// NETWORK 2
fbCase_DuplicateUpdateToDB(
    bExecute := bExecute,
    bUseInterimCodeForValidation := bUseInterimCodeForValidation,
    aOCVPackStatus := aOCVPackStatus,
    aOuterStatus := aOuterStatus,
    stOCVDataDB := stOCVDataDB,
    stOACDataDB := stOACDataDB,
    stOuterBarcodeDuplicate := stOuterBarcodeDuplicate,
    stOuterDuplicatedPackCodesFound := stOuterDuplicatedPackCodesFound,
    stCodeInfo_Pack := stCodeInfo_Pack,
    stCodeInfo_Intermediate := stCodeInfo_Intermediate,
    stCodeInfo_Outer := stCodeInfo_Outer,
    stCACData := stCACData,
    bBusy => bBusy,
    bError => bError,
    nErrorID => nErrorID,
    nOACFilesBlocked => nOACFilesBlocked,
    nOCVFilesBlocked => nOCVFilesBlocked,
    stDaigOACDataDB => stDaigOACDataDB,
    stDiagOCVDataDB => stDiagOCVDataDB); // FB_CASE_DuplicateUpdateToDB
bDone := fbCase_DuplicateUpdateToDB.bDone;

ACTION Init:

rTrigDataInit(CLK := bDataInit);

IF rTrigDataInit.Q THEN
	
	stProductInstruction.nOutersPerCase		:= 50;
	stProductInstruction.nPacksPerOuter 	:= 10;
	
	stCACData.NumberOfOuters	:= 50;
	

	FOR iOuter := 1 TO stProductInstruction.nOutersPerCase DO
		(* Ustaw outer *)
		stCACData.Outer[iOuter].Barcode    := CONCAT('OUTER', INT_TO_STRING(iOuter));
		stCACData.Outer[iOuter].OuterCodeStatus := 5;
		
		stCACData.Outer[iOuter].OuterRejectID	:= 0;
		
		
		FOR iPack := 1 TO stProductInstruction.nPacksPerOuter DO
			(* Pack number z zerami *)
			sPackNum := CONCAT('0', INT_TO_STRING(iPack));  (* dla 1-9: '01'-'09' *)
			IF iPack = 10 THEN
				sPackNum := '10';
			END_IF;
			
			(* Outer number z zerami dla 1-9 *)
			sOuterNum := CONCAT('0', INT_TO_STRING(iOuter));
			IF iOuter >= 10 THEN
				sOuterNum := INT_TO_STRING(iOuter);
			END_IF;
			
			(* Sklej pack code *)
			sPackCode := CONCAT(CONCAT('PACK', sPackNum), CONCAT('OUTER', sOuterNum));
			
			(* Przypisz *)
			stCACData.Outer[iOuter].PackCode[iPack]			:= sPackCode;
			stCACData.Outer[iOuter].PackCodeStatus[iPack]	:= 5;
			stCACData.Outer[iOuter].PackRejectID[iPack]		:= 0;
			
		END_FOR;
	END_FOR;	
	
END_IF
END_ACTION

END_PROGRAM

// ---- POUs/FinaliseCaseData/FB_CASE_DuplicateUpdateToDB.TcPOU
(* reads CAC files from CAC folder, deletes OAC file and copies CAC file into Archive *)
FUNCTION_BLOCK FB_CASE_DuplicateUpdateToDB
VAR_INPUT
	bExecute				: BOOL;		(* set TRUE to archive OAC files *)
	bUseInterimCodeForValidation	: BOOL;
END_VAR
VAR_IN_OUT
	
	aOCVPackStatus			: ARRAY[1..cMAX_OUTER_STATUS_QUEUE] OF ST_OUTER_Status;	(* Outer status array *)
	aOuterStatus				: ARRAY[1..cMAX_OUTER_STATUS_QUEUE] OF ST_OUTER_Status;	(* Outer status array *)
	
	//stProductInstruction		: ST_PCM_Status;
	stOCVDataDB				: ST_DB_OCVDataCtrl;
	stOACDataDB				: ST_DB_OACDataCtrl;
	
	stOuterBarcodeDuplicate			: ST_RejectItems;
	stOuterDuplicatedPackCodesFound	: ST_RejectItems;
	
	stCodeInfo_Pack			: ST_CodeInfo;
	stCodeInfo_Intermediate	: ST_CodeInfo;
	stCodeInfo_Outer		: ST_CodeInfo;
	
	stCACData			: ST_CAC_Data;
END_VAR
VAR_OUTPUT
	bDone 					: BOOL;		(* TRUE = OAC archive complete *)
	bBusy 					: BOOL;		(* TRUE = OAC archive active *)
	bError 					: BOOL;		(* TRUE = OAC archive error *)
	nErrorID				: UDINT;	(* error code *)

	nOACFilesBlocked		: UINT;
	nOCVFilesBlocked		: UINT;
	stDaigOACDataDB				: ST_DB_OACDataCtrl;
	stDiagOCVDataDB				: ST_DB_OCVDataCtrl;
	

END_VAR
VAR
	fbExecute				: R_TRIG;
	eState					: E_CAC_State;
	eErrorState				: E_CAC_State;

	tonTimeOut				: TON;
	rtTimeOutExec			: R_TRIG;
	
	stOCVStatus				: ST_OUTER_Status;
	stOACStatus				: ST_OUTER_Status;
	
	nOuterIndex				: INT;
	nOACIndex				: INT;
	nOCVIndex				: INT;
END_VAR

(***************************************TimeOut *******************************************)
(* monitor Busy timeout *)
tonTimeOut( IN:=bBusy, PT:=cTEN_SECONDS, Q=>);
(*	cTHREE_SECONDS						: TIME := T#3s;
	cFIVE_SECONDS						: TIME := t#5s;
	cTEN_SECONDS						: TIME := t#10s;*)

rtTimeOutExec(CLK:= tonTimeOut.Q);

IF rtTimeOutExec.Q THEN

	bError := TRUE;
	nErrorID := 100;
	eErrorState := eState;

	MEMSET(ADR(stOCVDataDB), 16#00, SIZEOF(stOCVDataDB));
	MEMSET(ADR(stOACDataDB), 16#00, SIZEOF(stOACDataDB));

	eState := E_CAC_DONE;
END_IF

(***************************************Execution*******************************************)

(* monitor bExecute for rising edge *)
fbExecute(CLK := bExecute);

CASE eState OF

	(* idle *)
	E_CAC_IDLE:

		(* rising edge of bExecute *)
		IF fbExecute.Q = TRUE THEN

			(* update outputs *)
			bDone := FALSE;
			bBusy := TRUE;
			bError := FALSE;
			nErrorID := 0;

			
			MEMSET(ADR(stOCVDataDB), 16#00, SIZEOF(stOCVDataDB));
			MEMSET(ADR(stOACDataDB), 16#00, SIZEOF(stOACDataDB));

			nOACFilesBlocked 	:= 0;
			nOCVFilesBlocked 	:= 0;

			nOuterIndex			:= 1;
			
			eState := E_CAC_DUPLICATEOUTERCHECK;

		(* bExecute has been reset *)
		ELSIF bExecute = FALSE THEN

			(* clear outputs *)
			bDone := FALSE;
			bBusy := FALSE;
			bError := FALSE;
			(*nErrorID := 0;*)
		END_IF

(*****************************************************************************************)

	(* check outer reject code for dupicate found*)
	E_CAC_DUPLICATEOUTERCHECK:

		IF stCACData.Outer[nOuterIndex].OuterRejectID = stOuterDuplicatedPackCodesFound.nRejectID OR 
			stCACData.Outer[nOuterIndex].OuterRejectID = stOuterBarcodeDuplicate.nRejectID THEN
		
			FillInDBData();
	
			stOACDataDB.bBlockRecord			:= TRUE;
			stOCVDataDB.bBlockRecord			:= TRUE;
			
			stOACDataDB.bUpdateDataReq			:= TRUE;
			stOCVDataDB.bUpdateDataReq			:= TRUE;
			
			eState := E_CAC_DELETEOAC;
		ELSE
			IF nOuterIndex = stCACData.NumberOfOuters THEN

				eState := E_CAC_DONE;
			ELSE
				nOuterIndex := LIMIT(1, nOuterIndex + 1, stCACData.NumberOfOuters);
			END_IF
		END_IF

	(* delete OAC files *)
	E_CAC_DELETEOAC:

		FOR nOACIndex := 1 TO cMAX_OUTER_STATUS_QUEUE DO
			IF aOuterStatus[nOACIndex].stOACData.Barcode =  stOACDataDB.stOACStatusDB.stOACData.Barcode AND 
				aOuterStatus[nOACIndex].stOACData.Barcode <> '' THEN

				//MEMSET(ADR(aOuterStatus[nOACIndex].stOACData), 16#00, SIZEOF(aOuterStatus[nOACIndex].stOACData));
				aOuterStatus[nOACIndex].nStatus.22 := TRUE;
				aOuterStatus[nOACIndex].stOACData.DataSource := 'REM';
			END_IF
		END_FOR

		IF	stOACDataDB.bDone	THEN

			IF NOT  stOACDataDB.bError THEN

				nOACFilesBlocked := nOACFilesBlocked + 1;
			ELSE
				bError := TRUE;
				nErrorID := stOACDataDB.nErrorID;
				eErrorState := eState;
			END_IF
			stDaigOACDataDB := stOACDataDB;
			MEMSET(ADR(stOACDataDB), 16#00, SIZEOF(stOACDataDB));

			eState := E_CAC_DELETEOCV1;
		END_IF

	E_CAC_DELETEOCV1:

		IF stOCVDataDB.stOCVStatusDB.stOACData.AggregationCodes[1] <> '' 	OR 
			stOCVDataDB.stOCVStatusDB.stOACData.AggregationCodes[2] <> '' 	THEN

			FOR nOCVIndex := 1 TO cMAX_OUTER_STATUS_QUEUE DO
				IF aOCVPackStatus[nOCVIndex].stOACData.AggregationCodes[1] =  stOCVDataDB.stOCVStatusDB.stOACData.AggregationCodes[1] 	AND
					aOCVPackStatus[nOCVIndex].stOACData.AggregationCodes[2] =  stOCVDataDB.stOCVStatusDB.stOACData.AggregationCodes[2]	THEN
					
					//MEMSET(ADR(aOCVPackStatus[nOCVIndex].stOACData), 16#00, SIZEOF(aOCVPackStatus[nOCVIndex].stOACData));
					aOCVPackStatus[nOCVIndex].nStatus.22 := TRUE;
					aOCVPackStatus[nOCVIndex].stOACData.DataSource := 'REM';
				END_IF
			END_FOR
		END_IF
		
		IF	stOCVDataDB.bDone	THEN

			IF NOT  stOCVDataDB.bError THEN

				nOCVFilesBlocked := nOCVFilesBlocked + 1;
			ELSE
				bError := TRUE;
				nErrorID := stOCVDataDB.nErrorID;
				eErrorState := eState;
			END_IF

			stDiagOCVDataDB := stOCVDataDB;
			MEMSET(ADR(stOCVDataDB), 16#00, SIZEOF(stOCVDataDB));
			
			IF nOuterIndex = stCACData.NumberOfOuters THEN

				eState := E_CAC_DONE;
			ELSE
				nOuterIndex := LIMIT(1, nOuterIndex + 1, stCACData.NumberOfOuters);
				
				eState := E_CAC_DUPLICATEOUTERCHECK;
			END_IF
		END_IF

	(* complete *)
	E_CAC_DONE:

		(* update outputs *)
		bBusy := FALSE;
		bDone := TRUE;

		eState := E_CAC_IDLE;

(* unknown state *)
ELSE

	eState := E_CAC_IDLE;
END_CASE

ACTION FillInDBData:
(************************************************************Fill In OAC Data****************************************************************************)

IF F_InvalidateASCIIChar(F_CODE_GetItem(stCACData.Outer[nOuterIndex].Barcode, eCodeAIType.SerialCode, stCodeInfo_Outer)) >	0 	THEN

	stOACDataDB.sFileCodeName	:='';
ELSE
	stOACDataDB.sFileCodeName	:= F_CodeToHex(F_CODE_GetItem(stCACData.Outer[nOuterIndex].Barcode , eCodeAIType.SerialCode, stCodeInfo_Outer));
END_IF

stOACDataDB.stOACStatusDB.stOACData	:= stCACData.Outer[nOuterIndex];
stOACDataDB.stOACStatusDB.stOACData.DataSource := 'REM';
stOACDataDB.stOACStatusDB.nTriggerID :=9999;
stOACDataDB.stOACStatusDB.nStatus.22 := TRUE;
stOACDataDB.stOACStatusDB.sDataSourceTracker := 'Dup Update';

FOR nOCVindex :=1 TO stOACDataDB.stOACStatusDB.stOACData.NumberOfPacks DO

	IF	stOACDataDB.stOACStatusDB.stOACData.PackCodeStatus[nOCVindex].5  THEN
		stOACDataDB.stOACStatusDB.aOACPackStatus[nOCVindex] :=5;
	ELSIF stOACDataDB.stOACStatusDB.stOACData.PackCodeStatus[nOCVindex].3  THEN
		stOACDataDB.stOACStatusDB.aOACPackStatus[nOCVindex] :=3;
	ELSE
		stOACDataDB.stOACStatusDB.aOACPackStatus[nOCVindex] :=0;
	END_IF
END_FOR

(************************************************************Fill In OCV Data****************************************************************************)


IF F_InvalidateASCIIChar(F_CODE_GetItem(stCACData.Outer[nOuterIndex].AggregationCodes[1] , eCodeAIType.SerialCode,
										SEL(bUseInterimCodeForValidation, stCodeInfo_Pack, stCodeInfo_Intermediate))) >	0 	THEN

	stOCVDataDB.sFileCodeName1	:= '';
ELSE
	stOCVDataDB.sFileCodeName1	:= F_CodeToHex(F_CODE_GetItem(stCACData.Outer[nOuterIndex].AggregationCodes[1] , eCodeAIType.SerialCode,
																		SEL(bUseInterimCodeForValidation, stCodeInfo_Pack, stCodeInfo_Intermediate)));
END_IF

IF F_InvalidateASCIIChar(F_CODE_GetItem(stCACData.Outer[nOuterIndex].AggregationCodes[2] , eCodeAIType.SerialCode,   stCodeInfo_Pack)) >	0 	THEN

	stOCVDataDB.sFileCodeName2	:='';
ELSE
	stOCVDataDB.sFileCodeName2	:= F_CodeToHex(F_CODE_GetItem(stCACData.Outer[nOuterIndex].AggregationCodes[2] , eCodeAIType.SerialCode,   stCodeInfo_Pack));
END_IF

stOCVDataDB.stOCVStatusDB.stOACData	:= stCACData.Outer[nOuterIndex];
stOCVDataDB.stOCVStatusDB.stOACData.DataSource := 'REM';
stOCVDataDB.stOCVStatusDB.nTriggerID :=9999;
stOCVDataDB.stOCVStatusDB.nStatus.22 := TRUE;
stOCVDataDB.stOCVStatusDB.sDataSourceTracker	:= 'Dup Update';

FOR nOCVindex :=1 TO stOCVDataDB.stOCVStatusDB.stOACData.NumberOfPacks DO

	IF	stOCVDataDB.stOCVStatusDB.stOACData.PackCodeStatus[nOCVindex].5  THEN
		stOCVDataDB.stOCVStatusDB.aOACPackStatus[nOCVindex] :=5;
	ELSIF stOCVDataDB.stOCVStatusDB.stOACData.PackCodeStatus[nOCVindex].3  THEN
		stOCVDataDB.stOCVStatusDB.aOACPackStatus[nOCVindex] :=3;
	ELSE
		stOCVDataDB.stOCVStatusDB.aOACPackStatus[nOCVindex] :=0;
	END_IF
END_FOR
END_ACTION

END_FUNCTION_BLOCK

// ---- POUs/_Utilites/METS/F_InvalidateASCIIChar.TcPOU
FUNCTION F_InvalidateASCIIChar : INT
VAR_INPUT
	sCode		: STRING(255);
END_VAR
VAR
	nCodeLen	: INT;
	nCharIndex		: INT;
	sChar			: STRING(1);
END_VAR

(* reset output *)
F_InvalidateASCIIChar := 0;

(* strPackCode contains data *)
IF LEN(sCode) = 0 THEN

	F_InvalidateASCIIChar := -1;

ELSIF LEN(sCode) > 0 THEN

	(* check each char in the code *)
	FOR nCharIndex := 1 TO LEN(sCode) DO

		(* get char from string *)
		sChar := MID(sCode, 1, nCharIndex);

		(* check if every char valid for proccessig*)
		IF (F_ToASC(sChar) < 16#21 OR  F_ToASC(sChar) >  16#7A) AND   F_ToASC(sChar) <> 16#7C THEN	(*  16#7C -> '|'*)

			(* update valid char counter *)
			F_InvalidateASCIIChar := F_InvalidateASCIIChar + 1;
		END_IF
	END_FOR
END_IF

END_FUNCTION

// ---- POUs/_Utilites/METS/F_CODE_GetItem.TcPOU
FUNCTION F_CODE_GetItem : T_MaxString
VAR_INPUT
	sFullCode			: T_MaxString;
	nCodeType		: INT;
	stCodeInfo		: ST_CodeInfo;
END_VAR
VAR
	stItem			: ST_CodeValidation;
	eCodeAIPattern	: E_CodeAIType;
	sItem			: T_MaxString;
	nStart			: INT;
	nEnd				: INT;
	sTemp			: T_MaxString;
END_VAR

IF stCodeInfo.nEntireLength > 0 THEN

	IF nCodeType = eCodeAIPattern.GTIN THEN 				stItem := stCodeInfo.stGTIN;
	ELSIF nCodeType = eCodeAIPattern.BatchID THEN 		stItem := stCodeInfo.stBatchID;
	ELSIF nCodeType = eCodeAIPattern.SerialCode THEN		stItem := stCodeInfo.stSerialCode;
	ELSIF nCodeType = eCodeAIPattern.ProductionOrder THEN	stItem := stCodeInfo.stProductionOrder;
	ELSIF nCodeType = eCodeAIPattern.CryptoCode THEN		stItem := stCodeInfo.stCryptoCode;
	ELSIF nCodeType = eCodeAIPattern.RSKU THEN			stItem := stCodeInfo.stRSKU;
	ELSIF nCodeType = eCodeAIPattern.MRP THEN			stItem := stCodeInfo.stMRP;
	ELSIF nCodeType = eCodeAIPattern.BrandSpecification THEN		stItem := stCodeInfo.stBrandSpecification;
	ELSIF nCodeType = eCodeAIPattern.ProduceDate THEN		stItem := stCodeInfo.stProduceDate;
	ELSIF nCodeType = eCodeAIPattern.UserField3 THEN		stItem := stCodeInfo.stUserField3;
	END_IF


	IF stItem.sStartAI <> '' AND stItem.sEndAI <> '' THEN
		nStart := FIND(sFullCode, stItem.sStartAI) + LEN(stItem.sStartAI);
		IF nStart > 0 THEN
			sTemp := RIGHT(sFullCode, LEN(sFullCode) - (nStart - 1));
		ELSE
			sTemp := sFullCode;
		END_IF
		nEnd := FIND(sTemp, stItem.sEndAI);
		IF nEnd = 0 THEN
			nEnd := LEN(sFullCode)+1;
		ELSE
			nEnd := nEnd +(nStart - 1);
		END_IF
	ELSIF stItem.sStartAI <> '' AND stItem.nCodeLength > 0 THEN
		nStart := FIND(sFullCode, stItem.sStartAI) + LEN(stItem.sStartAI);
		nEnd := nStart + stItem.nCodeLength;
	ELSIF stItem.nCodeStartPos > 0 AND stItem.sEndAI <> '' THEN
		nStart := stItem.nCodeStartPos;
		sTemp := RIGHT(sFullCode, LEN(sFullCode) - (nStart - 1));
		nEnd := FIND(sTemp, stItem.sEndAI);
		IF nEnd = 0 THEN
			nEnd := LEN(sFullCode)+1;
		ELSE
			nEnd := nEnd +(nStart - 1);
		END_IF
	ELSIF stItem.nCodeStartPos >= 0 AND stItem.nCodeLength > 0 THEN
		nStart := stItem.nCodeStartPos;
		nEnd := nStart + stItem.nCodeLength;
	ELSE
		nStart := 0;
		nEnd := 0;
	END_IF
	IF nStart > 0 AND nEnd > 0 THEN
		sItem := MID(sFullCode, nEnd - nStart, nStart);
	ELSE
		sItem := '';
	END_IF
ELSE
	sItem := '';
END_IF

F_CODE_GetItem := sItem;

END_FUNCTION

// ---- POUs/TcUnit/FB_CASE_FinaliseDataTests/PRG_CASE_FinaliseDataManual.TcPOU
PROGRAM PRG_CASE_FinaliseDataManual
VAR
	fbCase_FinaliseData		: FB_CASE_FinaliseData;
	
	(* Init function/method declarations*)
	rTrigDataInit		: R_TRIG;
	bDataInit			: BOOL;
	iOuter				: INT;
	iPack				: INT;
	sPackNum			: STRING;
	sOuterNum			: STRING;
	sPackCode			: STRING;
	
	(* Inputs *)
	bExecute 				: BOOL;		(* set TRUE to move Outers *)
	bDoorReject				: BOOL;
	stRejectReasonsForCase	: ST_RejectReasonsForCase;
	
	(* In/Out *)
	stProductInstruction	: ST_PCM_Status;
	stCodeInfo_Outer		: ST_CodeInfo;
	stCACData 				: ST_CAC_Data;	(* Case Queue *)
	stCACDataHMI			: ST_HMI_CAC_Data;
	
	(* Outputs *)
	bDone 					: BOOL;
	bBusy					: BOOL;

	bCACValid				: BOOL;
	bCACInvalid				: BOOL;

	bCheckDuplicates		: BOOL;
	bReadyToValidate		: BOOL;
	
	sRejectCode				: T_MaxString;
	sCaseContent			: T_LongSTRING;
	
END_VAR

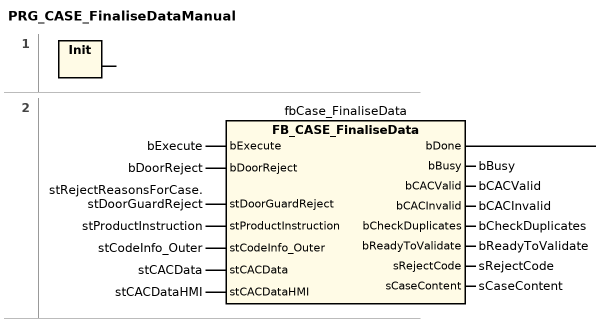
// NETWORK 1
Init();

// NETWORK 2
fbCase_FinaliseData(
    bExecute := bExecute,
    bDoorReject := bDoorReject,
    stDoorGuardReject := stRejectReasonsForCase.stDoorGuardReject,
    stProductInstruction := stProductInstruction,
    stCodeInfo_Outer := stCodeInfo_Outer,
    stCACData := stCACData,
    stCACDataHMI := stCACDataHMI,
    bBusy => bBusy,
    bCACValid => bCACValid,
    bCACInvalid => bCACInvalid,
    bCheckDuplicates => bCheckDuplicates,
    bReadyToValidate => bReadyToValidate,
    sRejectCode => sRejectCode,
    sCaseContent => sCaseContent); // FB_CASE_FinaliseData

ACTION Init:

rTrigDataInit(CLK := bDataInit);

IF rTrigDataInit.Q THEN
	
stProductInstruction.nOutersPerCase		:= 50;
stProductInstruction.nPacksPerOuter 	:= 10;

	FOR iOuter := 1 TO stProductInstruction.nOutersPerCase DO
		(* Outer number z zerami *)
		sOuterNum := F_StringAddPrefix(INT_TO_STRING(iOuter),2,'0');
		
		(* Write Outers barcodes *)
		stCACData.Outer[iOuter].Barcode    := CONCAT('OUTER', sOuterNum);
		stCACData.Outer[iOuter].OuterCodeStatus := 5;
		stCACData.Outer[iOuter].OuterRejectCode := 'OK';
		
		FOR iPack := 1 TO stProductInstruction.nPacksPerOuter DO
			(* Pack number dwucyfrowy z zerami *)
			sPackNum := F_StringAddPrefix(INT_TO_STRING(iPack),2,'0');			
			(* Sklej pack code *)
			sPackCode := CONCAT(CONCAT('PACK', sPackNum), CONCAT('OUTER', sOuterNum));
			
			(* Write Pack Barcodes / Data*)
			stCACData.Outer[iOuter].PackCode[iPack]			:= sPackCode;
			stCACData.Outer[iOuter].PackCodeStatus[iPack]	:= 5;
			stCACData.Outer[iOuter].PackRejectID[iPack]		:= 0;			
			stCACData.Outer[iOuter].PackRejectCode[iPack]	:= 'OK';
			
						
			stCACData.Outer[iOuter].NumberOfPacks := stProductInstruction.nPacksPerOuter;
			
		END_FOR;
	END_FOR;	

//initialize needed data structures
stCACData.NumberOfOuters						:= stProductInstruction.nOutersPerCase;
stCACData.CaseRejectCode						:= 'OK';
stCodeInfo_Outer.nEntireLength					:= 7;
stCodeInfo_Outer.stSerialCode.nCodeStartPos 	:= 1;
stCodeInfo_Outer.stSerialCode.nCodeLength 		:= 7;
stCACData.Barcode 								:= 'CaseBarcode';
	
END_IF
END_ACTION

END_PROGRAM

// ---- POUs/FinaliseCaseData/FB_CASE_FinaliseData.TcPOU
FUNCTION_BLOCK FB_CASE_FinaliseData
VAR_INPUT
	bExecute 			: BOOL;		(* set TRUE to move Outers *)
	//stCTDateTime			: ST_SYSTEM_DateTime;
	bDoorReject				: BOOL;
	stDoorGuardReject		: ST_RejectItems;
END_VAR
VAR_IN_OUT
	stProductInstruction	: ST_PCM_Status;
	stCodeInfo_Outer		: ST_CodeInfo;
	stCACData 				: ST_CAC_Data;	(* Case Queue *)
	stCACDataHMI			: ST_HMI_CAC_Data;

END_VAR
VAR_OUTPUT
	bDone 					: BOOL;
	bBusy					: BOOL;

	bCACValid			: BOOL;
	bCACInvalid			: BOOL;

	bCheckDuplicates		: BOOL;
	bReadyToValidate		: BOOL;
	
	sRejectCode				: T_MaxString;
	sCaseContent			: T_LongSTRING;
END_VAR
VAR
	rtExecute				: R_TRIG;
	
	nOuterIndex				: INT;
	nPackIndex				: INT;
	
	sAppendedString			: T_MaxString;
	nCaseContentLogIndex	: INT;
END_VAR

(* rising edge of bExecute *)
rtExecute(CLK:= bExecute);

(* validate stCACData *)
IF rtExecute.Q THEN

	(* clear outputs *)
	bCACValid 				:= FALSE;
	bCACInvalid 			:= FALSE;

	bCheckDuplicates		:= FALSE;
	bReadyToValidate		:= FALSE;
	sRejectCode 	:= '';

	IF bDoorReject THEN

		stCACData.CaseRejectCode 	:= stDoorGuardReject.sMetsDisplayCode;
		stCACData.CaseRejectID 		:= stDoorGuardReject.nRejectID;
	END_IF
	
(******************************************************************************************************************************************)
	(* clear HMI data *)
	MEMSET(ADR(stCACDataHMI), 16#00, SIZEOF(stCACDataHMI));

	(*copy data to stCaseQueueHMI[1]*)
	IF stCACData.CaseRejectCode = 'OK' THEN
		
		(* CAC data is valid *)
		bCACValid := TRUE;
		bCACInvalid := FALSE;
		
		stCACDataHMI.sBarcode:= F_CONCAT3(stCACData.Barcode,'(999)','1');
	ELSE
		(* CAC data is invalid *)
		bCACValid := FALSE;
		bCACInvalid := TRUE;
		
		stCACDataHMI.sBarcode:= F_CONCAT3(stCACData.Barcode,'(999)','0');
	END_IF

	stCACDataHMI.nNumberOfOuters 	:= stCACData.NumberOfOuters;
	stCACDataHMI.nNumberOfPacks 	:= stCACData.Outer[1].NumberOfPacks;

	FOR nOuterIndex:=1 TO MIN(stCACData.NumberOfOuters, cMAX_OUTERS_PER_CASE) DO
		
		IF stCACData.Outer[nOuterIndex].OuterRejectCode = 'OK' THEN
			stCACDataHMI.aOuter[nOuterIndex].sBarcode:= F_CONCAT3(stCACData.Outer[nOuterIndex].Barcode,'(999)','1');
		ELSE
			stCACDataHMI.aOuter[nOuterIndex].sBarcode:= F_CONCAT3(stCACData.Outer[nOuterIndex].Barcode,'(999)','0');
		END_IF

		FOR nPackIndex:=1 TO MIN(stCACData.Outer[nOuterIndex].NumberOfPacks, cMAX_PACKS_PER_OUTER) DO
			IF stCACData.Outer[nOuterIndex].PackRejectCode[nPackIndex] = 'OK' THEN
				stCACDataHMI.aOuter[nOuterIndex].aPackCode[nPackIndex]:= F_CONCAT3(stCACData.Outer[nOuterIndex].PackCode[nPackIndex],'(999)','1');
			ELSE
				stCACDataHMI.aOuter[nOuterIndex].aPackCode[nPackIndex]:= F_CONCAT3(stCACData.Outer[nOuterIndex].PackCode[nPackIndex],'(999)','0');
			END_IF
		END_FOR
	END_FOR

(******************************************************************************************************************************************)

	sAppendedString	:= '';
	sCaseContent 	:= '';
	
	sCaseContent := F_CONCAT3(' [', INT_TO_STRING(stCACData.NumberOfOuters),']:');
	FOR nCaseContentLogIndex := 1 TO MIN(stCACData.NumberOfOuters ,cMAX_OUTERS_PER_CASE) BY 1 DO
		//sCaseContent :=F_LongCONCAT(sCaseContent, '   ');
		//sCaseContent := F_LongCONCAT(sCaseContent, RIGHT(F_CODE_GetItem(stCACData.Outer[nCaseContentLogIndex].Barcode, eCodeAIType.SerialCode,  stCodeInfo_Outer),7));
	
		CONCAT2(ADR(sCaseContent), ADR('   '), ADR(sCaseContent), SIZEOF(sCaseContent));
	
		sAppendedString := RIGHT(F_CODE_GetItem(stCACData.Outer[nCaseContentLogIndex].Barcode, eCodeAIType.SerialCode,  stCodeInfo_Outer),7);
		CONCAT2(ADR(sCaseContent), ADR(sAppendedString), ADR(sCaseContent), SIZEOF(sCaseContent));
	END_FOR

(******************************************************************************************************************************************)

	sRejectCode 	:= stCACData.CaseRejectCode;
	bDone := TRUE;

(* bExecute has been reset *)
ELSIF bExecute = FALSE THEN

	bDone := FALSE;

END_IF

END_FUNCTION_BLOCK

// ---- POUs/TcUnit/FB_CASE_InitialiseData/PRG_CASE_InitialiseDataManual.TcPOU
PROGRAM PRG_CASE_InitialiseDataManual
VAR
	fbCase_InitialiseData		: FB_CASE_InitialiseData;
	
	(* Init function/method declarations*)
	rTrigDataInit		: R_TRIG;
	bDataInit			: BOOL;
	iOuter				: INT;
	iPack				: INT;
	sPackNum			: STRING;
	sOuterNum			: STRING;
	sPackCode			: STRING;
	
	// old variables
	nOuterIndex				: INT;
	nPackIndex				: INT;
	
	(* Inputs *)	
	bExecute 				: BOOL;	(* set TRUE to move Outers *)
	stCTDateTime			: ST_SYSTEM_DateTime;
	stRejectReasonsForCase	: ST_RejectReasonsForCase;
	
	
	(* In/Out *)
	stProductInstruction	: ST_PCM_Status := (sFieldName := 'PCM_Status_name', nOutersPerCase := 50);
	stCACData 				: ST_CAC_Data;	(* Case Queue *)
	
	(* Outputs *)
	bDone					: BOOL;
	bBusy					: BOOL;
	bDoorReject				: BOOL;
	sRejectCode				: T_MaxString;		
	nMasterListCounter		: INT;	
	bCheckDuplicates		: BOOL;
	
END_VAR

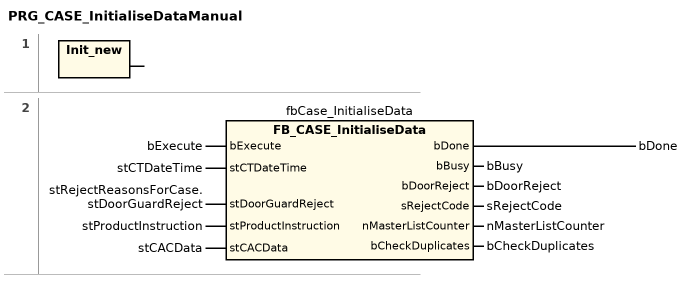
// NETWORK 1
Init_new();

// NETWORK 2
fbCase_InitialiseData(
    bExecute := bExecute,
    stCTDateTime := stCTDateTime,
    stDoorGuardReject := stRejectReasonsForCase.stDoorGuardReject,
    stProductInstruction := stProductInstruction,
    stCACData := stCACData,
    bBusy => bBusy,
    bDoorReject => bDoorReject,
    sRejectCode => sRejectCode,
    nMasterListCounter => nMasterListCounter,
    bCheckDuplicates => bCheckDuplicates); // FB_CASE_InitialiseData
bDone := fbCase_InitialiseData.bDone;

ACTION Init:

rTrigDataInit(CLK := bDataInit);

IF rTrigDataInit.Q THEN
	
	MEMSET(ADR(stCACData), 16#00, SIZEOF(stCACData));	
	
	stProductInstruction.nOutersPerCase 	:= 50;
	stProductInstruction.nPacksPerOuter		:= 10;
	stProductInstruction.nOpMode			:= 11;
	stProductInstruction.sRetailSKU			:= '1234567';
	stProductInstruction.nAcceptanceLevel 	:= 10;


	stCACData.NumberOfOuters			:= stProductInstruction.nOutersPerCase;
	stCACData.CodingAndTrackingMode		:= stProductInstruction.nOpMode;
	stCACData.RetailSKU					:= stProductInstruction.sRetailSKU;

	FOR nOuterIndex := 1 TO stProductInstruction.nOutersPerCase BY 1 DO
	
	stCACData.Outer[nOuterIndex].Barcode 					:= CONCAT('OUTER_', INT_TO_STRING(nOuterIndex));
	stCACData.Outer[nOuterIndex].NumberOfPacks 				:= stProductInstruction.nPacksPerOuter;
	stCACData.Outer[nOuterIndex].NumberOfLinkedPacks 		:= stProductInstruction.nPacksPerOuter;
	stCACData.Outer[nOuterIndex].AcceptanceLevel 			:= stProductInstruction.nAcceptanceLevel;
	stCACData.Outer[nOuterIndex].CodingAndTrackingMode		:= stProductInstruction.nOpMode;
	stCACData.Outer[nOuterIndex].OuterRejectCode			:= 'OK';
	
		FOR  nPackIndex :=1 TO stProductInstruction.nPacksPerOuter BY 1 DO
			stCACData.Outer[nOuterIndex].PackCode[nPackIndex] 		:= F_CONCAT3(stCACData.Outer[nOuterIndex].Barcode,'_PACK_', INT_TO_STRING(nPackIndex));
			IF nPackIndex = 1 THEN
				stCACData.Outer[nOuterIndex].AggregationCodes[1]	:= stCACData.Outer[nOuterIndex].PackCode[nPackIndex];
			END_IF
			IF nPackIndex = 2 THEN
				stCACData.Outer[nOuterIndex].AggregationCodes[2]	:= stCACData.Outer[nOuterIndex].PackCode[nPackIndex];
			END_IF
			stCACData.Outer[nOuterIndex].PackCodeStatus[nPackIndex].5 	:= TRUE;
			stCACData.Outer[nOuterIndex].PackRejectCode[nPackIndex]		:= 'OK';
		END_FOR
	END_FOR	
	
	stCACData.Outer[3].OuterCodeStatus.5 	:= TRUE;
	stCACData.Outer[4].OuterCodeStatus.5	:= TRUE;
	
END_IF
END_ACTION

ACTION Init_new:

rTrigDataInit(CLK := bDataInit);

IF rTrigDataInit.Q THEN
	
	MEMSET(ADR(stCACData), 16#00, SIZEOF(stCACData));	
	
	stProductInstruction.nOutersPerCase 	:= 50;
	stProductInstruction.nPacksPerOuter		:= 10;
	stProductInstruction.nOpMode			:= 11;
	stProductInstruction.sRetailSKU			:= '1234567';
	stProductInstruction.nAcceptanceLevel 	:= 10;


	stCACData.NumberOfOuters			:= stProductInstruction.nOutersPerCase;
	stCACData.CodingAndTrackingMode		:= stProductInstruction.nOpMode;
	stCACData.RetailSKU					:= stProductInstruction.sRetailSKU;

	FOR iOuter := 1 TO stProductInstruction.nOutersPerCase DO
		(* Outer number z zerami *)
		sOuterNum := F_StringAddPrefix(INT_TO_STRING(iOuter),2,'0');
	
		stCACData.Outer[iOuter].Barcode    				:= CONCAT('OUTER', sOuterNum);
		stCACData.Outer[iOuter].NumberOfPacks 			:= stProductInstruction.nPacksPerOuter;
		stCACData.Outer[iOuter].NumberOfLinkedPacks 	:= stProductInstruction.nPacksPerOuter;
		stCACData.Outer[iOuter].AcceptanceLevel 		:= stProductInstruction.nAcceptanceLevel;
		stCACData.Outer[iOuter].CodingAndTrackingMode	:= stProductInstruction.nOpMode;
		stCACData.Outer[iOuter].OuterRejectCode			:= 'OK';
	
		FOR iPack := 1 TO stProductInstruction.nPacksPerOuter DO
			(* Pack number dwucyfrowy z zerami *)
			sPackNum := F_StringAddPrefix(INT_TO_STRING(iPack),2,'0');			
			(* Sklej pack code *)
			sPackCode := CONCAT(CONCAT('PACK', sPackNum), CONCAT('OUTER', sOuterNum));
			
			(* Write Pack Barcodes / Data*)
			stCACData.Outer[iOuter].PackCode[iPack]				:= sPackCode;
			stCACData.Outer[iOuter].PackCodeStatus[iPack]		:= 5;
			stCACData.Outer[iOuter].PackRejectID[iPack]			:= 0;			
			stCACData.Outer[iOuter].PackRejectCode[iPack]		:= 'OK';			
			stCACData.Outer[iOuter].PackCodeStatus[iPack].5 	:= TRUE;
			
			
			IF iPack = 1 THEN
				stCACData.Outer[iOuter].AggregationCodes[1]	:= stCACData.Outer[iOuter].PackCode[iPack];
			END_IF
			IF iPack = 2 THEN
				stCACData.Outer[iOuter].AggregationCodes[2]	:= stCACData.Outer[iOuter].PackCode[iPack];
			END_IF
		END_FOR
	END_FOR	
	
	stCACData.Outer[3].OuterCodeStatus.5 	:= TRUE;
	stCACData.Outer[4].OuterCodeStatus.5	:= TRUE;
	
END_IF
END_ACTION

END_PROGRAM

// ---- POUs/FinaliseCaseData/FB_CASE_InitialiseData.TcPOU
FUNCTION_BLOCK FB_CASE_InitialiseData
VAR_INPUT
	bExecute 			: BOOL;		(* set TRUE to move Outers *)
	stCTDateTime			: ST_SYSTEM_DateTime;
	stDoorGuardReject		: ST_RejectItems;
END_VAR
VAR_IN_OUT
	stProductInstruction	: ST_PCM_Status;
	stCACData 				: ST_CAC_Data;	(* Case Queue *)
END_VAR
VAR_OUTPUT
	bDone 					: BOOL;
	bBusy					: BOOL;

	bDoorReject				: BOOL;
	sRejectCode				: T_MaxString;
	nMasterListCounter		: INT;
	
	bCheckDuplicates		: BOOL;
	
END_VAR
VAR
	rtExecute				: R_TRIG;
	nOuterIndex				: INT;
END_VAR

(* rising edge of bExecute *)
rtExecute(CLK:= bExecute);

		(* validate stCACData *)
IF rtExecute.Q THEN

	bDoorReject			:= FALSE;
	nMasterListCounter	:=0;
	sRejectCode 		:= '';
	bCheckDuplicates	:= FALSE;
	
	(* populate case data *)
	(* date (YYYY-MM-DD) and time (hh:mm:ss) with offset to UTC *)
	stCACData.ProductionDate 		:= F_StringWildcard('#YYYYMMDD#', stCTDateTime.sSystemTime);
	stCACData.ProductionTime 		:= F_StringWildcard('#hhmmss#', stCTDateTime.sSystemTime);
	stCACData.ProductionTimeOffset 	:= F_SYSTEM_SystemTimeOffsetToHHMM(stCTDateTime.nSystemTimeOffset);

	(* product and machine info *)
	stCACData.RetailSKU 				:= stProductInstruction.sRetailSKU;    (*sCPIData.RetailSKU;*)
	stCACData.CasePacker.ProductionSite := stProductInstruction.sProductionSite; (*sCPIData.ProductionSite  ;*)
	stCACData.CasePacker.ProductionLine := stProductInstruction.sProductionLine;  (*   sCPIData.ProductionLine;*)
	stCACData.CodingAndTrackingMode 	:= stProductInstruction.nOpMode;  (*STRING_TO_INT(sCPIData.CodingAndTrackingMode);*)

	(* PassThrough, PrePrintedLabel or PrintApply mode active *)
	IF stCACData.CodingAndTrackingMode <= 6 THEN

		(* non-aggregated case, populate NumberOfOuters and CodingAndTrackingMode *)
		stCACData.NumberOfOuters := stProductInstruction.nOutersPerCase;

		//stCACData.CaseRejectCode := 'OK';
		//stCACData.CaseRejectID := 0;

	(* CaseTrace or PackTrace mode *)
	ELSE
		FOR nOuterIndex := 1 TO stProductInstruction.nOutersPerCase DO
			
			IF stCACData.Outer[nOuterIndex].OuterMasterListRestored THEN
				nMasterListCounter := nMasterListCounter +1;
			END_IF
			
			IF stCACData.Outer[nOuterIndex].OuterCodeStatus.5 AND stCACData.NumberOfOuters = stProductInstruction.nOutersPerCase  THEN
				stCACData.NumberOfOuters := -3;		//b5		Outer Code - Val Index error found
			END_IF
		END_FOR
		
		stCACData.CaseRejectCode := 'OK';
		stCACData.CaseRejectID := 0;
		
	END_IF
	
	IF stCACData.CaseRejectID =	stDoorGuardReject.nRejectID THEN
		bDoorReject	:= TRUE;
	END_IF

	sRejectCode 		:= stCACData.CaseRejectCode;
	bCheckDuplicates	:= TRUE;
	bDone 				:= TRUE;
		
(* bExecute has been reset *)
ELSIF bExecute = FALSE THEN

	bDone := FALSE;

END_IF

END_FUNCTION_BLOCK

// ---- POUs/TcUnit/FB_CASE_ValidateContentTests/PRG_CASE_ValidateContentManual.TcPOU
PROGRAM PRG_CASE_ValidateContentManual
VAR
	fbCase_ValidateContent		: FB_CASE_ValidateContent;
	
	
	(* Init function/method declarations*)
	rTrigDataInit		: R_TRIG;
	bDataInit			: BOOL;
	iOuter				: INT;
	iPack				: INT;
	sPackNum			: STRING;
	sOuterNum			: STRING;
	sPackCode			: STRING;
	
	(* Inputs *)
	bExecute 					: BOOL;
	stCTDateTime				: ST_SYSTEM_DateTime;	(* CaseTrace date/time structure *)
	
	(* In/Out *)
	stProductInstruction		: ST_PCM_Status;
	nSecquentionalCounter		: UDINT;
	stCodeInfo_Outer			: ST_CodeInfo;
	stCaseRejectReasons			: ST_RejectReasonsForCase;
	stCACData 					: ST_CAC_Data;
	
	(* Outputs *)
	bDone 						: BOOL;
	bBusy						: BOOL;
	bError						: BOOL;
	nErrorID 					: UDINT;

	sRejectCode					: T_MaxString;
	nValidationIndex			: INT;
	
END_VAR

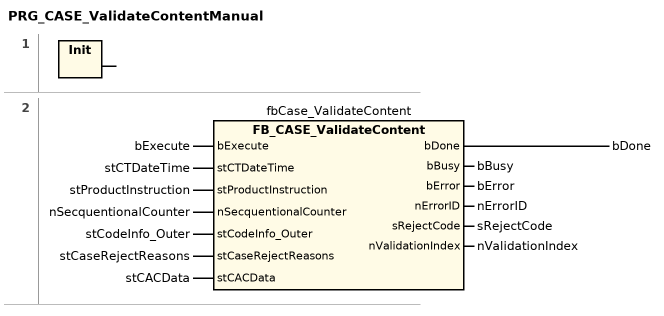
// NETWORK 1
Init();

// NETWORK 2
fbCase_ValidateContent(
    bExecute := bExecute,
    stCTDateTime := stCTDateTime,
    stProductInstruction := stProductInstruction,
    nSecquentionalCounter := nSecquentionalCounter,
    stCodeInfo_Outer := stCodeInfo_Outer,
    stCaseRejectReasons := stCaseRejectReasons,
    stCACData := stCACData,
    bBusy => bBusy,
    bError => bError,
    nErrorID => nErrorID,
    sRejectCode => sRejectCode,
    nValidationIndex => nValidationIndex); // FB_CASE_ValidateContent
bDone := fbCase_ValidateContent.bDone;

ACTION Init:

rTrigDataInit(CLK := bDataInit);

IF rTrigDataInit.Q THEN
	
stProductInstruction.nOutersPerCase		:= 50;
stProductInstruction.nPacksPerOuter 	:= 10;

	FOR iOuter := 1 TO stProductInstruction.nOutersPerCase DO
		(* Ustaw outer *)
		stCACData.Outer[iOuter].Barcode    := CONCAT('OUTER', INT_TO_STRING(iOuter));
		stCACData.Outer[iOuter].OuterCodeStatus := 5;
		
		FOR iPack := 1 TO stProductInstruction.nPacksPerOuter DO
			(* Pack number z zerami *)
			sPackNum := CONCAT('0', INT_TO_STRING(iPack));  (* dla 1-9: '01'-'09' *)
			IF iPack = 10 THEN
				sPackNum := '10';
			END_IF;
			
			(* Outer number z zerami dla 1-9 *)
			sOuterNum := CONCAT('0', INT_TO_STRING(iOuter));
			IF iOuter >= 10 THEN
				sOuterNum := INT_TO_STRING(iOuter);
			END_IF;
			
			(* Sklej pack code *)
			sPackCode := CONCAT(CONCAT('PACK', sPackNum), CONCAT('OUTER', sOuterNum));
			
			(* Przypisz *)
			stCACData.Outer[iOuter].PackCode[iPack]			:= sPackCode;
			stCACData.Outer[iOuter].PackCodeStatus[iPack]	:= 5;
			stCACData.Outer[iOuter].PackRejectID[iPack]		:= 0;
			
		END_FOR;
	END_FOR;	
	
END_IF
END_ACTION

END_PROGRAM

// ---- POUs/FBReferenceTest/FB_TimersTEST.TcPOU
FUNCTION_BLOCK FB_TimersTEST
VAR_INPUT
	bStartTON	: BOOL;
	bStartTOF	: BOOL;
	tTime		: TIME;
END_VAR

VAR_IN_OUT	
	tTON			: TON;
	tTOF			: TOF;
END_VAR

VAR_OUTPUT
	tTON_Q		: BOOL;
	tTOF_Q		: BOOL;
END_VAR
VAR
	tPTton			: TIME;
	tPTtof			: TIME;
	
END_VAR


tPTtof := tTime;
tPTton := tTime;

tTON(IN := bStartTON, PT := tPTton, Q => tTON_Q);
tTOF(IN := bStartTOF, PT := tPTtof, Q => tTOF_Q);

END_FUNCTION_BLOCK

// ---- POUs/FBReferenceTest/PRG_Reference_POU.TcPOU
PROGRAM PRG_Reference_POU
VAR
	
	fbTimersTEST	: FB_TimersTEST;
	
	tTON_Q			: BOOL;
	tTOF_Q			: BOOL;
	
	tTimer			: TIME := T#4S;
	
	bStartTON		: BOOL;
	bStartTOF		: BOOL;
	
	
END_VAR


fbTimersTEST(
	bStartTON:= bStartTON, 
	bStartTOF:= bStartTOF, 
	tTime:= tTimer, 
	tTON:= GVL_test.stFBinside.aTONs[1],
	tTOF:= GVL_test.stFBinside.aTOFs[1],
	tTON_Q=> tTON_Q, 
	tTOF_Q=> tTOF_Q
);

END_PROGRAM

// ---- POUs/FinaliseCaseData/FB_CASE_MovePackerToCase.TcPOU
(* move Outers up to and including strOuterBarcode from aPackerQueue  to stCACData *)
FUNCTION_BLOCK FB_CASE_MovePackerToCase
VAR_INPUT
	bExecute 				: BOOL;		(* set TRUE to move Outers *)
	stDoorGuardReject		: ST_RejectItems;
END_VAR
VAR_IN_OUT
	stProductInstruction	: ST_PCM_Status;
	aPackerQueue			: ARRAY [0..1] OF ST_CASE_InfeedQueue;
	stCACData 				: ST_CAC_Data;	(* Case Queue *)
END_VAR
VAR_OUTPUT
	bDone 					: BOOL;		(* TRUE = complete *)
	bDoorReject				: BOOL;
	nNumberOfOuters			: INT;
	sFirstBarcodeInCase		: T_OUTER_Barcode;
	sLastBarcodeInCase		: T_OUTER_Barcode;
END_VAR
VAR
	fbExecute				: R_TRIG;
	nOuterIndex				: INT;

END_VAR

(* rising edge of bExecute *)
fbExecute(CLK:= bExecute);

(* move CaseData *)
IF fbExecute.Q = TRUE THEN

	//nMaxOuterIndex := UDINT_TO_INT(SIZEOF(stCaseQueue.aCACData[1].Outer) / SIZEOF(stCaseQueue.aCACData[1].Outer[1]));

	(* clear data *)
	bDoorReject	:= FALSE;
	MEMSET(ADR(stCACData.Outer), 16#00, SIZEOF(stCACData.Outer));

	stCACData.NumberOfOuters:= aPackerQueue[0].nIndex + aPackerQueue[1].nIndex;

	IF stCACData.NumberOfOuters <= cMAX_OUTERS_PER_CASE THEN
	(* shift specified*)
		MEMMOVE(ADR(stCACData.Outer[1]), ADR(aPackerQueue[1].aOuter), SIZEOF(aPackerQueue[1].aOuter[1]) * F_SafeTo_UDINT(aPackerQueue[1].nIndex));
		MEMMOVE(ADR(stCACData.Outer[aPackerQueue[1].nIndex + 1]), ADR(aPackerQueue[0].aOuter), SIZEOF(aPackerQueue[0].aOuter[1]) * F_SafeTo_UDINT(aPackerQueue[0].nIndex));

		nNumberOfOuters	:= 	stCACData.NumberOfOuters;
		sFirstBarcodeInCase	:=	stCACData.Outer[1].Barcode;
		sLastBarcodeInCase 	:=	stCACData.Outer[nNumberOfOuters].Barcode;
		
		IF stCACData.NumberOfOuters = stProductInstruction.nOutersPerCase THEN
			FOR nOuterIndex := 1 TO stCACData.NumberOfOuters DO
				IF stCACData.Outer[nOuterIndex].OuterCodeStatus.5 THEN
					stCACData.NumberOfOuters := -3;		//b5		Outer Code - Val Index error found
				END_IF
			END_FOR
		END_IF
		
	ELSE
		stCACData.NumberOfOuters := -1;			// Outers number exceed cMAX_OUTERS_PER_CASE 

		nNumberOfOuters	:= 	stCACData.NumberOfOuters;
		sFirstBarcodeInCase	:=	'';
		sLastBarcodeInCase 	:=	'';
	END_IF

	IF aPackerQueue[0].bDoorReject OR aPackerQueue[1].bDoorReject THEN
		
		stCACData.CaseRejectCode := stDoorGuardReject.sMetsDisplayCode;
		stCACData.CaseRejectID := stDoorGuardReject.nRejectID;
		bDoorReject	:= TRUE;
	END_IF

	(* clear data *)
	MEMSET(ADR(aPackerQueue), 16#00, SIZEOF(aPackerQueue));
	
	bDone := TRUE;

(* bExecute has been reset *)
ELSIF bExecute = FALSE THEN
	bDone := FALSE;
END_IF

END_FUNCTION_BLOCK

// ---- POUs/TcUnit/FB_CASE_DuplicatCheckTests/FB_CASE_DuplicatCheckTests.TcPOU
FUNCTION_BLOCK FB_CASE_DuplicatCheckTests EXTENDS TcUnit.FB_TestSuite

VAR
	
	(* In/Out test*)
	stProductInstruction_tests					: ST_PCM_Status;
	stOuterBarcodeDuplicate_tests				: ST_RejectItems;
	stOuterDuplicatedPackCodesFound_tests		: ST_RejectItems;
	stCaseRejectReasons_tests					: ST_RejectReasonsForCase;		
	stRejectReasonForOuters_tests				: ST_RejectReasonsForOuter;	
	stRejectReasonForPacks_tests				: ST_RejectReasonsForPack;	
	
	stCACData_tests 							: ST_CAC_Data;	
	stUpdateCACData_tests						: ST_CAC_Data;	
	sRejectCode_tests							: T_MaxString;

	
END_VAR

		
stProductInstruction_tests.nOutersPerCase		:= 50;
stProductInstruction_tests.nPacksPerOuter 		:= 10;

//==============================================================
//01.Main
//==============================================================

//main02_bIsDuplicatePackTRUEonPackBarcodeDuplicate();
//main03_OuterRejectIDChangedWhenOuterDuplicate();

//==============================================================
//02.OuterDuplicate
//==============================================================
OuterDuplicate01_bIsDuplicateOuterTRUEonOuterBarcodeDuplicate();
OuterDuplicate02_bIsDuplicateOuterTRUEonOuterBarcodeDuplicate();
OuterDuplicate03_bIsDuplicateOuterTRUEonOuterBarcodeDuplicate();
OuterDuplicate04_bIsDuplicateOuterTRUEonOuterBarcodeDuplicate();
OuterDuplicate05_bIsDuplicateOuterTRUEonOuterBarcodeDuplicate();

//==============================================================
//03.OuterBarcodeEmpty
//==============================================================
OuterBarcodeEmpty01_OneOuterBarcodeEmptyNoDuplicatFound();
OuterBarcodeEmpty02_TwoOutersBarcodeEmptyNoDuplicatFound();


//==============================================================
//04.PackDuplicate
//==============================================================
PackDuplicate01_bIsDuplicatePacksTRUEonPackBarcodeDuplicate();
PackDuplicate02_bIsDuplicatePacksTRUEonPackBarcodeDuplicateWithinSameOuter();

//==============================================================
//05.PackBarcodeEmpty
//==============================================================
PackBarcodeEmpty01_OnePackBarcodeEmpty();
PackBarcodeEmpty02_TwoPackBarcodeEmptyDifferentOuters();
PackBarcodeEmpty03_TwoPackBarcodeEmptySameOuter();

//==============================================================
//06.bCACValidStatus
//==============================================================
bCACValidStatus01_FALSEOnOuterBarcodeDuplicate();
bCACValidStatus02_FALSEOn2OuterBarcodeDuplicate();
bCACValidStatus03_FALSEOnSeveralOutersBarcodeDuplicate();
bCACValidStatus04_FALSEOn2PackBarcodeDuplicate();
bCACValidStatus05_FALSEOn2PacksSameOuterBarcodeDuplicate();

//==============================================================
//07.sRejectCodeString
//==============================================================
sRejectCodeString01_WrongValueOn1OuterDuplicate();
sRejectCodeString02_WrongValueOn2PacksDuplicateIn1Outer();
sRejectCodeString03_WrongValueOn2PacksDuplicateIn2Outers();
sRejectCodeString04_WrongValueOnSeveralOutersDuplicate();
sRejectCodeString05_WrongValueOnSeveralPacksDuplicateInSeveralOuters();

METHOD INTERNAL bCACValidStatus01_FALSEOnOuterBarcodeDuplicate
VAR
	fbCase_tests					: FB_CASE_DuplicatCheck;
	
	
	bDone_tests 					: BOOL;
	bBusy_tests						: BOOL;

	bCACValid_tests					: BOOL;
	bIsDuplicateOuter_tests			: BOOL;
	bIsDuplicatePacks_tests			: BOOL;
	
	bReadyToValidate_tests			: BOOL;
	
END_VAR

//Data initialization
TestInit(stCACData:= stCACData_tests, stProductInstruction:= stProductInstruction_tests);

//Change some data for test scenario below
stCACData_tests.Outer[1].Barcode := stCACData_tests.Outer[10].Barcode;

	
TcUnit.TEST('bCACValidStatus01_FALSEOnOuterBarcodeDuplicate');

fbCase_tests(
	bExecute:= TRUE, 
	stProductInstruction:= stProductInstruction_tests, 
	stPackCodesDuplicated:= stRejectReasonForOuters_tests.stOuterDuplicatedPackCodesFound, 
	stOuterBarcodeDuplicate:= stRejectReasonForOuters_tests.stOuterBarcodeDuplicate, 
	stOuterDuplicatedPackCodesFound:= stRejectReasonForOuters_tests.stOuterDuplicatedPackCodesFound, 
	stCaseRejectReasons:= stCaseRejectReasons_tests, 
	stCACData:= stCACData_tests, 
	bDone=> bDone_tests, 
	bBusy=> bBusy_tests, 
	bCACValid=> bCACValid_tests, 
	sRejectCode=> sRejectCode_tests, 
	bIsDuplicateOuters=> bIsDuplicateOuter_tests, 
	bIsDuplicatePacks=> bIsDuplicatePacks_tests, 
	bReadyToValidate=> bReadyToValidate_tests, 
	stUpdateCACData=> stUpdateCACData_tests
);

	
AssertEquals_BOOL( Expected	:= FALSE,
			 	   Actual	:= bCACValid_tests, 
			 	   Message	:= 'Wrong bCACVAlid value on outer duplicate');
						

TEST_FINISHED();
END_METHOD

METHOD INTERNAL bCACValidStatus02_FALSEOn2OuterBarcodeDuplicate
VAR
	fbCase_tests					: FB_CASE_DuplicatCheck;
	
	
	bDone_tests 					: BOOL;
	bBusy_tests						: BOOL;

	bCACValid_tests					: BOOL;
	bIsDuplicateOuter_tests			: BOOL;
	bIsDuplicatePacks_tests			: BOOL;
	
	bReadyToValidate_tests			: BOOL;
	
END_VAR

//Data initialization
TestInit(stCACData:= stCACData_tests, stProductInstruction:= stProductInstruction_tests);

//Change some data for test scenario below
stCACData_tests.Outer[1].Barcode := stCACData_tests.Outer[10].Barcode;
stCACData_tests.Outer[8].Barcode := stCACData_tests.Outer[34].Barcode;

	
TcUnit.TEST('bCACValidStatus02_FALSEOn2OuterBarcodeDuplicate');

fbCase_tests(
	bExecute:= TRUE, 
	stProductInstruction:= stProductInstruction_tests, 
	stPackCodesDuplicated:= stRejectReasonForOuters_tests.stOuterDuplicatedPackCodesFound, 
	stOuterBarcodeDuplicate:= stRejectReasonForOuters_tests.stOuterBarcodeDuplicate, 
	stOuterDuplicatedPackCodesFound:= stRejectReasonForOuters_tests.stOuterDuplicatedPackCodesFound, 
	stCaseRejectReasons:= stCaseRejectReasons_tests, 
	stCACData:= stCACData_tests, 
	bDone=> bDone_tests, 
	bBusy=> bBusy_tests, 
	bCACValid=> bCACValid_tests, 
	sRejectCode=> sRejectCode_tests, 
	bIsDuplicateOuters=> bIsDuplicateOuter_tests, 
	bIsDuplicatePacks=> bIsDuplicatePacks_tests, 
	bReadyToValidate=> bReadyToValidate_tests, 
	stUpdateCACData=> stUpdateCACData_tests
);

	
AssertEquals_BOOL( Expected	:= FALSE,
			 	   Actual	:= bCACValid_tests, 
			 	   Message	:= 'Wrong bCACVAlid value on outer duplicate');
						

TEST_FINISHED();
END_METHOD

METHOD INTERNAL bCACValidStatus03_FALSEOnSeveralOutersBarcodeDuplicate
VAR
	fbCase_tests					: FB_CASE_DuplicatCheck;
	
	
	bDone_tests 					: BOOL;
	bBusy_tests						: BOOL;

	bCACValid_tests					: BOOL;
	bIsDuplicateOuter_tests			: BOOL;
	bIsDuplicatePacks_tests			: BOOL;
	
	bReadyToValidate_tests			: BOOL;
	
END_VAR

//Data initialization
TestInit(stCACData:= stCACData_tests, stProductInstruction:= stProductInstruction_tests);

//Change some data for test scenario below
stCACData_tests.Outer[1].Barcode := stCACData_tests.Outer[5].Barcode;
stCACData_tests.Outer[6].Barcode := stCACData_tests.Outer[11].Barcode;
stCACData_tests.Outer[12].Barcode := stCACData_tests.Outer[18].Barcode;
stCACData_tests.Outer[19].Barcode := stCACData_tests.Outer[24].Barcode;
stCACData_tests.Outer[27].Barcode := stCACData_tests.Outer[31].Barcode;

	
TcUnit.TEST('bCACValidStatus03_FALSEOnSeveralOutersBarcodeDuplicate');

fbCase_tests(
	bExecute:= TRUE, 
	stProductInstruction:= stProductInstruction_tests, 
	stPackCodesDuplicated:= stRejectReasonForOuters_tests.stOuterDuplicatedPackCodesFound, 
	stOuterBarcodeDuplicate:= stRejectReasonForOuters_tests.stOuterBarcodeDuplicate, 
	stOuterDuplicatedPackCodesFound:= stRejectReasonForOuters_tests.stOuterDuplicatedPackCodesFound, 
	stCaseRejectReasons:= stCaseRejectReasons_tests, 
	stCACData:= stCACData_tests, 
	bDone=> bDone_tests, 
	bBusy=> bBusy_tests, 
	bCACValid=> bCACValid_tests, 
	sRejectCode=> sRejectCode_tests, 
	bIsDuplicateOuters=> bIsDuplicateOuter_tests, 
	bIsDuplicatePacks=> bIsDuplicatePacks_tests, 
	bReadyToValidate=> bReadyToValidate_tests, 
	stUpdateCACData=> stUpdateCACData_tests
);

	
AssertEquals_BOOL( Expected	:= FALSE,
			 	   Actual	:= bCACValid_tests, 
			 	   Message	:= 'Wrong bCACVAlid value on outer duplicate');
						

TEST_FINISHED();
END_METHOD

METHOD INTERNAL bCACValidStatus04_FALSEOn2PackBarcodeDuplicate
VAR
	fbCase_tests					: FB_CASE_DuplicatCheck;
	
	
	bDone_tests 					: BOOL;
	bBusy_tests						: BOOL;

	bCACValid_tests					: BOOL;
	bIsDuplicateOuter_tests			: BOOL;
	bIsDuplicatePacks_tests			: BOOL;
	
	bReadyToValidate_tests			: BOOL;
	
END_VAR

//Data initialization
TestInit(stCACData:= stCACData_tests, stProductInstruction:= stProductInstruction_tests);

//Change some data for test scenario below
stCACData_tests.Outer[7].PackCode[4] := stCACData_tests.Outer[28].PackCode[7];

	
TcUnit.TEST('bCACValidStatus04_FALSEOn2PackBarcodeDuplicate');

fbCase_tests(
	bExecute:= TRUE, 
	stProductInstruction:= stProductInstruction_tests, 
	stPackCodesDuplicated:= stRejectReasonForOuters_tests.stOuterDuplicatedPackCodesFound, 
	stOuterBarcodeDuplicate:= stRejectReasonForOuters_tests.stOuterBarcodeDuplicate, 
	stOuterDuplicatedPackCodesFound:= stRejectReasonForOuters_tests.stOuterDuplicatedPackCodesFound, 
	stCaseRejectReasons:= stCaseRejectReasons_tests, 
	stCACData:= stCACData_tests, 
	bDone=> bDone_tests, 
	bBusy=> bBusy_tests, 
	bCACValid=> bCACValid_tests, 
	sRejectCode=> sRejectCode_tests, 
	bIsDuplicateOuters=> bIsDuplicateOuter_tests, 
	bIsDuplicatePacks=> bIsDuplicatePacks_tests, 
	bReadyToValidate=> bReadyToValidate_tests, 
	stUpdateCACData=> stUpdateCACData_tests
);

	
AssertEquals_BOOL( Expected	:= FALSE,
			 	   Actual	:= bCACValid_tests, 
			 	   Message	:= 'Wrong bCACVAlid value on outer duplicate');
						

TEST_FINISHED();
END_METHOD

METHOD INTERNAL bCACValidStatus05_FALSEOn2PacksSameOuterBarcodeDuplicate
VAR
	fbCase_tests					: FB_CASE_DuplicatCheck;
	
	
	bDone_tests 					: BOOL;
	bBusy_tests						: BOOL;

	bCACValid_tests					: BOOL;
	bIsDuplicateOuter_tests			: BOOL;
	bIsDuplicatePacks_tests			: BOOL;
	
	bReadyToValidate_tests			: BOOL;
	
END_VAR

//Data initialization
TestInit(stCACData:= stCACData_tests, stProductInstruction:= stProductInstruction_tests);

//Change some data for test scenario below
stCACData_tests.Outer[12].PackCode[1] := stCACData_tests.Outer[12].PackCode[9];

	
TcUnit.TEST('bCACValidStatus05_FALSEOn2PacksSameOuterBarcodeDuplicate');

fbCase_tests(
	bExecute:= TRUE, 
	stProductInstruction:= stProductInstruction_tests, 
	stPackCodesDuplicated:= stRejectReasonForOuters_tests.stOuterDuplicatedPackCodesFound, 
	stOuterBarcodeDuplicate:= stRejectReasonForOuters_tests.stOuterBarcodeDuplicate, 
	stOuterDuplicatedPackCodesFound:= stRejectReasonForOuters_tests.stOuterDuplicatedPackCodesFound, 
	stCaseRejectReasons:= stCaseRejectReasons_tests, 
	stCACData:= stCACData_tests, 
	bDone=> bDone_tests, 
	bBusy=> bBusy_tests, 
	bCACValid=> bCACValid_tests, 
	sRejectCode=> sRejectCode_tests, 
	bIsDuplicateOuters=> bIsDuplicateOuter_tests, 
	bIsDuplicatePacks=> bIsDuplicatePacks_tests, 
	bReadyToValidate=> bReadyToValidate_tests, 
	stUpdateCACData=> stUpdateCACData_tests
);

	
AssertEquals_BOOL( Expected	:= FALSE,
			 	   Actual	:= bCACValid_tests, 
			 	   Message	:= 'Wrong bCACVAlid value on outer duplicate');
						

TEST_FINISHED();
END_METHOD

METHOD INTERNAL main02_bIsDuplicatePackTRUEonPackBarcodeDuplicate
VAR
	fbCase					: FB_CASE_DuplicatCheck;
	bIsDuplicateOuter		: BOOL;
	bIsDuplicatePacks		: BOOL;
	

	
END_VAR

//Data initialization
TestInit(stCACData:= stCACData_tests, stProductInstruction:= stProductInstruction_tests);

//Change some data for test scenario below
stCACData_tests.Outer[9].PackCode[2] := stCACData_tests.Outer[15].PackCode[5];

	
TcUnit.TEST('main02_bIsDuplicatePackTRUEonPackBarcodeDuplicate');

// fbCase(
// 	bExecute:= TRUE, 
// 	stProductInstruction:= , 
// 	stPackCodesDuplicated:= , 
// 	stOuterBarcodeDuplicate:= , 
// 	stOuterDuplicatedPackCodesFound:= , 
// 	stCaseRejectReasons:= , 
// 	stCACData:= , 
// 	bDone=> , 
// 	bBusy=> , 
// 	bCACValid=> , 
// 	sRejectCode=> , 
// 	bIsDuplicateOuters=> , 
// 	bIsDuplicatePacks=> , 
// 	bReadyToValidate=> , 
// 	stUpdateCACData=> 
// );

	
AssertEquals_BOOL( Expected	:= TRUE,
			 	   Actual	:= bIsDuplicatePacks, 
			 	   Message	:= 'Duplicated Pack barcode not found');
						

TEST_FINISHED();
END_METHOD

METHOD INTERNAL main03_OuterRejectIDChangedWhenOuterDuplicate
VAR
	fbCase					: FB_CASE_DuplicatCheck;
	bIsDuplicateOuter		: BOOL;
	bIsDuplicatePacks		: BOOL;
	

	
END_VAR

//Data initialization
TestInit(stCACData:= stCACData_tests, stProductInstruction:= stProductInstruction_tests);

//Change some data for test scenario below
stCACData_tests.Outer[2].Barcode := stCACData_tests.Outer[49].Barcode;

	
TcUnit.TEST('main03_OuterRejectIDChangedWhenOuterDuplicate');

// fbCase(
// 	bExecute:= TRUE, 
// 	stProductInstruction:= , 
// 	stPackCodesDuplicated:= , 
// 	stOuterBarcodeDuplicate:= , 
// 	stOuterDuplicatedPackCodesFound:= , 
// 	stCaseRejectReasons:= stCaseRejectReasons_01, 
// 	stCACData:= stCACData_01, 
// 	bDone=> , 
// 	bBusy=> , 
// 	bCACValid=> , 
// 	sRejectCode=> , 
// 	bIsDuplicateOuters=> bIsDuplicateOuter, 
// 	bIsDuplicatePacks=> bIsDuplicatePacks, 
// 	bReadyToValidate=> , 
// 	stUpdateCACData=> stUpdateCACData_01
// );

	
AssertEquals_UINT(Expected := 206,
                  Actual := stCACData_tests.Outer[2].OuterRejectID,
                  Message := 'OuterRejectID not updated when duplicate outer barcode');
						

TEST_FINISHED();
END_METHOD

METHOD INTERNAL OuterBarcodeEmpty01_OneOuterBarcodeEmptyNoDuplicatFound
VAR
	fbCase_tests					: FB_CASE_DuplicatCheck;
	
	
	bDone_tests 					: BOOL;
	bBusy_tests						: BOOL;

	bCACValid_tests					: BOOL;
	bIsDuplicateOuter_tests			: BOOL;
	bIsDuplicatePacks_tests			: BOOL;
	
	bReadyToValidate_tests			: BOOL;
	
END_VAR

//Data initialization
TestInit(stCACData:= stCACData_tests, stProductInstruction:= stProductInstruction_tests);

//Change some data for test scenario below
stCACData_tests.Outer[1].Barcode := '';

	
TcUnit.TEST('OuterBarcodeEmpty01_OneOuterBarcodeEmptyNoDuplicatFound');

fbCase_tests(
	bExecute:= TRUE, 
	stProductInstruction:= stProductInstruction_tests, 
	stPackCodesDuplicated:= stRejectReasonForOuters_tests.stOuterDuplicatedPackCodesFound, 
	stOuterBarcodeDuplicate:= stRejectReasonForOuters_tests.stOuterBarcodeDuplicate, 
	stOuterDuplicatedPackCodesFound:= stRejectReasonForOuters_tests.stOuterDuplicatedPackCodesFound, 
	stCaseRejectReasons:= stCaseRejectReasons_tests, 
	stCACData:= stCACData_tests, 
	bDone=> bDone_tests, 
	bBusy=> bBusy_tests, 
	bCACValid=> bCACValid_tests, 
	sRejectCode=> sRejectCode_tests, 
	bIsDuplicateOuters=> bIsDuplicateOuter_tests, 
	bIsDuplicatePacks=> bIsDuplicatePacks_tests, 
	bReadyToValidate=> bReadyToValidate_tests, 
	stUpdateCACData=> stUpdateCACData_tests
);

	
AssertEquals_BOOL( Expected	:= FALSE,
			 	   Actual	:= bIsDuplicateOuter_tests, 
			 	   Message	:= 'Duplicated Outer barcode not found');
						

TEST_FINISHED();
END_METHOD

METHOD INTERNAL OuterBarcodeEmpty02_TwoOutersBarcodeEmptyNoDuplicatFound
VAR
	fbCase_tests					: FB_CASE_DuplicatCheck;
	
	
	bDone_tests 					: BOOL;
	bBusy_tests						: BOOL;

	bCACValid_tests					: BOOL;
	bIsDuplicateOuter_tests			: BOOL;
	bIsDuplicatePacks_tests			: BOOL;
	
	bReadyToValidate_tests			: BOOL;
	
END_VAR

//Data initialization
TestInit(stCACData:= stCACData_tests, stProductInstruction:= stProductInstruction_tests);

//Change some data for test scenario below
stCACData_tests.Outer[1].Barcode := '';

	
TcUnit.TEST('OuterBarcodeEmpty02_TwoOutersBarcodeEmptyNoDuplicatFound');

fbCase_tests(
	bExecute:= TRUE, 
	stProductInstruction:= stProductInstruction_tests, 
	stPackCodesDuplicated:= stRejectReasonForOuters_tests.stOuterDuplicatedPackCodesFound, 
	stOuterBarcodeDuplicate:= stRejectReasonForOuters_tests.stOuterBarcodeDuplicate, 
	stOuterDuplicatedPackCodesFound:= stRejectReasonForOuters_tests.stOuterDuplicatedPackCodesFound, 
	stCaseRejectReasons:= stCaseRejectReasons_tests, 
	stCACData:= stCACData_tests, 
	bDone=> bDone_tests, 
	bBusy=> bBusy_tests, 
	bCACValid=> bCACValid_tests, 
	sRejectCode=> sRejectCode_tests, 
	bIsDuplicateOuters=> bIsDuplicateOuter_tests, 
	bIsDuplicatePacks=> bIsDuplicatePacks_tests, 
	bReadyToValidate=> bReadyToValidate_tests, 
	stUpdateCACData=> stUpdateCACData_tests
);

	
AssertEquals_BOOL( Expected	:= FALSE,
			 	   Actual	:= bIsDuplicateOuter_tests, 
			 	   Message	:= 'Duplicated Outer barcode not found');
						

TEST_FINISHED();
END_METHOD

METHOD INTERNAL OuterDuplicate01_bIsDuplicateOuterTRUEonOuterBarcodeDuplicate
VAR
	fbCase_tests					: FB_CASE_DuplicatCheck;
	
	
	bDone_tests 					: BOOL;
	bBusy_tests						: BOOL;

	bCACValid_tests					: BOOL;
	bIsDuplicateOuter_tests			: BOOL;
	bIsDuplicatePacks_tests			: BOOL;
	
	bReadyToValidate_tests			: BOOL;
	
END_VAR

//Data initialization
TestInit(stCACData:= stCACData_tests, stProductInstruction:= stProductInstruction_tests);

//Change some data for test scenario below
stCACData_tests.Outer[1].Barcode := stCACData_tests.Outer[50].Barcode;

	
TcUnit.TEST('OuterDuplicate01_bIsDuplicateOuterTRUEonOuterBarcodeDuplicate');

fbCase_tests(
	bExecute:= TRUE, 
	stProductInstruction:= stProductInstruction_tests, 
	stPackCodesDuplicated:= stRejectReasonForOuters_tests.stOuterDuplicatedPackCodesFound, 
	stOuterBarcodeDuplicate:= stRejectReasonForOuters_tests.stOuterBarcodeDuplicate, 
	stOuterDuplicatedPackCodesFound:= stRejectReasonForOuters_tests.stOuterDuplicatedPackCodesFound, 
	stCaseRejectReasons:= stCaseRejectReasons_tests, 
	stCACData:= stCACData_tests, 
	bDone=> bDone_tests, 
	bBusy=> bBusy_tests, 
	bCACValid=> bCACValid_tests, 
	sRejectCode=> sRejectCode_tests, 
	bIsDuplicateOuters=> bIsDuplicateOuter_tests, 
	bIsDuplicatePacks=> bIsDuplicatePacks_tests, 
	bReadyToValidate=> bReadyToValidate_tests, 
	stUpdateCACData=> stUpdateCACData_tests
);

	
AssertEquals_BOOL( Expected	:= TRUE,
			 	   Actual	:= bIsDuplicateOuter_tests, 
			 	   Message	:= 'Duplicated Outer barcode not found');
						

TEST_FINISHED();
END_METHOD

METHOD INTERNAL OuterDuplicate02_bIsDuplicateOuterTRUEonOuterBarcodeDuplicate
VAR
	fbCase_tests					: FB_CASE_DuplicatCheck;
	
	
	bDone_tests 					: BOOL;
	bBusy_tests						: BOOL;

	bCACValid_tests					: BOOL;
	bIsDuplicateOuter_tests			: BOOL;
	bIsDuplicatePacks_tests			: BOOL;
	
	bReadyToValidate_tests			: BOOL;
	
END_VAR

//Data initialization
TestInit(stCACData:= stCACData_tests, stProductInstruction:= stProductInstruction_tests);

//Change some data for test scenario below
stCACData_tests.Outer[24].Barcode := stCACData_tests.Outer[25].Barcode;

	
TcUnit.TEST('OuterDuplicate02_bIsDuplicateOuterTRUEonOuterBarcodeDuplicate');

fbCase_tests(
	bExecute:= TRUE, 
	stProductInstruction:= stProductInstruction_tests, 
	stPackCodesDuplicated:= stRejectReasonForOuters_tests.stOuterDuplicatedPackCodesFound, 
	stOuterBarcodeDuplicate:= stRejectReasonForOuters_tests.stOuterBarcodeDuplicate, 
	stOuterDuplicatedPackCodesFound:= stRejectReasonForOuters_tests.stOuterDuplicatedPackCodesFound, 
	stCaseRejectReasons:= stCaseRejectReasons_tests, 
	stCACData:= stCACData_tests, 
	bDone=> bDone_tests, 
	bBusy=> bBusy_tests, 
	bCACValid=> bCACValid_tests, 
	sRejectCode=> sRejectCode_tests, 
	bIsDuplicateOuters=> bIsDuplicateOuter_tests, 
	bIsDuplicatePacks=> bIsDuplicatePacks_tests, 
	bReadyToValidate=> bReadyToValidate_tests, 
	stUpdateCACData=> stUpdateCACData_tests
);

	
AssertEquals_BOOL( Expected	:= TRUE,
			 	   Actual	:= bIsDuplicateOuter_tests, 
			 	   Message	:= 'Duplicated Outer barcode not found');
						

TEST_FINISHED();
END_METHOD

METHOD INTERNAL OuterDuplicate03_bIsDuplicateOuterTRUEonOuterBarcodeDuplicate
VAR
	fbCase_tests					: FB_CASE_DuplicatCheck;
	
	
	bDone_tests 					: BOOL;
	bBusy_tests						: BOOL;

	bCACValid_tests					: BOOL;
	bIsDuplicateOuter_tests			: BOOL;
	bIsDuplicatePacks_tests			: BOOL;
	
	bReadyToValidate_tests			: BOOL;
	
END_VAR

//Data initialization
TestInit(stCACData:= stCACData_tests, stProductInstruction:= stProductInstruction_tests);

//Change some data for test scenario below
stCACData_tests.Outer[1].Barcode := stCACData_tests.Outer[2].Barcode;

	
TcUnit.TEST('OuterDuplicate03_bIsDuplicateOuterTRUEonOuterBarcodeDuplicate');

fbCase_tests(
	bExecute:= TRUE, 
	stProductInstruction:= stProductInstruction_tests, 
	stPackCodesDuplicated:= stRejectReasonForOuters_tests.stOuterDuplicatedPackCodesFound, 
	stOuterBarcodeDuplicate:= stRejectReasonForOuters_tests.stOuterBarcodeDuplicate, 
	stOuterDuplicatedPackCodesFound:= stRejectReasonForOuters_tests.stOuterDuplicatedPackCodesFound, 
	stCaseRejectReasons:= stCaseRejectReasons_tests, 
	stCACData:= stCACData_tests, 
	bDone=> bDone_tests, 
	bBusy=> bBusy_tests, 
	bCACValid=> bCACValid_tests, 
	sRejectCode=> sRejectCode_tests, 
	bIsDuplicateOuters=> bIsDuplicateOuter_tests, 
	bIsDuplicatePacks=> bIsDuplicatePacks_tests, 
	bReadyToValidate=> bReadyToValidate_tests, 
	stUpdateCACData=> stUpdateCACData_tests
);

	
AssertEquals_BOOL( Expected	:= TRUE,
			 	   Actual	:= bIsDuplicateOuter_tests, 
			 	   Message	:= 'Duplicated Outer barcode not found');
						

TEST_FINISHED();
END_METHOD

METHOD INTERNAL OuterDuplicate04_bIsDuplicateOuterTRUEonOuterBarcodeDuplicate
VAR
	fbCase_tests					: FB_CASE_DuplicatCheck;
	
	
	bDone_tests 					: BOOL;
	bBusy_tests						: BOOL;

	bCACValid_tests					: BOOL;
	bIsDuplicateOuter_tests			: BOOL;
	bIsDuplicatePacks_tests			: BOOL;
	
	bReadyToValidate_tests			: BOOL;
	
END_VAR

//Data initialization
TestInit(stCACData:= stCACData_tests, stProductInstruction:= stProductInstruction_tests);

//Change some data for test scenario below
stCACData_tests.Outer[49].Barcode := stCACData_tests.Outer[50].Barcode;

	
TcUnit.TEST('OuterDuplicate04_bIsDuplicateOuterTRUEonOuterBarcodeDuplicate');

fbCase_tests(
	bExecute:= TRUE, 
	stProductInstruction:= stProductInstruction_tests, 
	stPackCodesDuplicated:= stRejectReasonForOuters_tests.stOuterDuplicatedPackCodesFound, 
	stOuterBarcodeDuplicate:= stRejectReasonForOuters_tests.stOuterBarcodeDuplicate, 
	stOuterDuplicatedPackCodesFound:= stRejectReasonForOuters_tests.stOuterDuplicatedPackCodesFound, 
	stCaseRejectReasons:= stCaseRejectReasons_tests, 
	stCACData:= stCACData_tests, 
	bDone=> bDone_tests, 
	bBusy=> bBusy_tests, 
	bCACValid=> bCACValid_tests, 
	sRejectCode=> sRejectCode_tests, 
	bIsDuplicateOuters=> bIsDuplicateOuter_tests, 
	bIsDuplicatePacks=> bIsDuplicatePacks_tests, 
	bReadyToValidate=> bReadyToValidate_tests, 
	stUpdateCACData=> stUpdateCACData_tests
);

	
AssertEquals_BOOL( Expected	:= TRUE,
			 	   Actual	:= bIsDuplicateOuter_tests, 
			 	   Message	:= 'Duplicated Outer barcode not found');
						

TEST_FINISHED();
END_METHOD

METHOD INTERNAL OuterDuplicate05_bIsDuplicateOuterTRUEonOuterBarcodeDuplicate
VAR
	fbCase_tests					: FB_CASE_DuplicatCheck;
	
	
	bDone_tests 					: BOOL;
	bBusy_tests						: BOOL;

	bCACValid_tests					: BOOL;
	bIsDuplicateOuter_tests			: BOOL;
	bIsDuplicatePacks_tests			: BOOL;
	
	bReadyToValidate_tests			: BOOL;
	
END_VAR

//Data initialization
TestInit(stCACData:= stCACData_tests, stProductInstruction:= stProductInstruction_tests);

//Change some data for test scenario below
stCACData_tests.Outer[22].Barcode := stCACData_tests.Outer[27].Barcode;

	
TcUnit.TEST('OuterDuplicate05_bIsDuplicateOuterTRUEonOuterBarcodeDuplicate');

fbCase_tests(
	bExecute:= TRUE, 
	stProductInstruction:= stProductInstruction_tests, 
	stPackCodesDuplicated:= stRejectReasonForOuters_tests.stOuterDuplicatedPackCodesFound, 
	stOuterBarcodeDuplicate:= stRejectReasonForOuters_tests.stOuterBarcodeDuplicate, 
	stOuterDuplicatedPackCodesFound:= stRejectReasonForOuters_tests.stOuterDuplicatedPackCodesFound, 
	stCaseRejectReasons:= stCaseRejectReasons_tests, 
	stCACData:= stCACData_tests, 
	bDone=> bDone_tests, 
	bBusy=> bBusy_tests, 
	bCACValid=> bCACValid_tests, 
	sRejectCode=> sRejectCode_tests, 
	bIsDuplicateOuters=> bIsDuplicateOuter_tests, 
	bIsDuplicatePacks=> bIsDuplicatePacks_tests, 
	bReadyToValidate=> bReadyToValidate_tests, 
	stUpdateCACData=> stUpdateCACData_tests
);

	
AssertEquals_BOOL( Expected	:= TRUE,
			 	   Actual	:= bIsDuplicateOuter_tests, 
			 	   Message	:= 'Duplicated Outer barcode not found');
						

TEST_FINISHED();
END_METHOD

METHOD INTERNAL PackBarcodeEmpty01_OnePackBarcodeEmpty
VAR
	fbCase_tests					: FB_CASE_DuplicatCheck;
	
	
	bDone_tests 					: BOOL;
	bBusy_tests						: BOOL;

	bCACValid_tests					: BOOL;
	bIsDuplicateOuter_tests			: BOOL;
	bIsDuplicatePacks_tests			: BOOL;
	
	bReadyToValidate_tests			: BOOL;
	
END_VAR

//Data initialization
TestInit(stCACData:= stCACData_tests, stProductInstruction:= stProductInstruction_tests);

//Change some data for test scenario below
stCACData_tests.Outer[1].PackCode[1] := '';

	
TcUnit.TEST('PackBarcodeEmpty01_OnePackBarcodeEmpty');

fbCase_tests(
	bExecute:= TRUE, 
	stProductInstruction:= stProductInstruction_tests, 
	stPackCodesDuplicated:= stRejectReasonForOuters_tests.stOuterDuplicatedPackCodesFound, 
	stOuterBarcodeDuplicate:= stRejectReasonForOuters_tests.stOuterBarcodeDuplicate, 
	stOuterDuplicatedPackCodesFound:= stRejectReasonForOuters_tests.stOuterDuplicatedPackCodesFound, 
	stCaseRejectReasons:= stCaseRejectReasons_tests, 
	stCACData:= stCACData_tests, 
	bDone=> bDone_tests, 
	bBusy=> bBusy_tests, 
	bCACValid=> bCACValid_tests, 
	sRejectCode=> sRejectCode_tests, 
	bIsDuplicateOuters=> bIsDuplicateOuter_tests, 
	bIsDuplicatePacks=> bIsDuplicatePacks_tests, 
	bReadyToValidate=> bReadyToValidate_tests, 
	stUpdateCACData=> stUpdateCACData_tests
);

	
AssertEquals_BOOL( Expected	:= FALSE,
			 	   Actual	:= bIsDuplicatePacks_tests, 
			 	   Message	:= 'Duplicated Pack barcode not found');
						

TEST_FINISHED();
END_METHOD

METHOD INTERNAL PackBarcodeEmpty02_TwoPackBarcodeEmptyDifferentOuters
VAR
	fbCase_tests					: FB_CASE_DuplicatCheck;
	
	
	bDone_tests 					: BOOL;
	bBusy_tests						: BOOL;

	bCACValid_tests					: BOOL;
	bIsDuplicateOuter_tests			: BOOL;
	bIsDuplicatePacks_tests			: BOOL;
	
	bReadyToValidate_tests			: BOOL;
	
END_VAR

//Data initialization
TestInit(stCACData:= stCACData_tests, stProductInstruction:= stProductInstruction_tests);

//Change some data for test scenario below
stCACData_tests.Outer[1].PackCode[1] := '';
stCACData_tests.Outer[2].PackCode[10] := '';

	
TcUnit.TEST('PackBarcodeEmpty02_TwoPackBarcodeEmptyDifferentOuters');

fbCase_tests(
	bExecute:= TRUE, 
	stProductInstruction:= stProductInstruction_tests, 
	stPackCodesDuplicated:= stRejectReasonForOuters_tests.stOuterDuplicatedPackCodesFound, 
	stOuterBarcodeDuplicate:= stRejectReasonForOuters_tests.stOuterBarcodeDuplicate, 
	stOuterDuplicatedPackCodesFound:= stRejectReasonForOuters_tests.stOuterDuplicatedPackCodesFound, 
	stCaseRejectReasons:= stCaseRejectReasons_tests, 
	stCACData:= stCACData_tests, 
	bDone=> bDone_tests, 
	bBusy=> bBusy_tests, 
	bCACValid=> bCACValid_tests, 
	sRejectCode=> sRejectCode_tests, 
	bIsDuplicateOuters=> bIsDuplicateOuter_tests, 
	bIsDuplicatePacks=> bIsDuplicatePacks_tests, 
	bReadyToValidate=> bReadyToValidate_tests, 
	stUpdateCACData=> stUpdateCACData_tests
);

	
AssertEquals_BOOL( Expected	:= FALSE,
			 	   Actual	:= bIsDuplicatePacks_tests, 
			 	   Message	:= 'Duplicated Pack barcode not found');
						

TEST_FINISHED();
END_METHOD

METHOD INTERNAL PackBarcodeEmpty03_TwoPackBarcodeEmptySameOuter
VAR
	fbCase_tests					: FB_CASE_DuplicatCheck;
	
	
	bDone_tests 					: BOOL;
	bBusy_tests						: BOOL;

	bCACValid_tests					: BOOL;
	bIsDuplicateOuter_tests			: BOOL;
	bIsDuplicatePacks_tests			: BOOL;
	
	bReadyToValidate_tests			: BOOL;
	
END_VAR

//Data initialization
TestInit(stCACData:= stCACData_tests, stProductInstruction:= stProductInstruction_tests);

//Change some data for test scenario below
stCACData_tests.Outer[3].PackCode[3] := '';
stCACData_tests.Outer[3].PackCode[5] := '';

	
TcUnit.TEST('PackBarcodeEmpty03_TwoPackBarcodeEmptySameOuter');

fbCase_tests(
	bExecute:= TRUE, 
	stProductInstruction:= stProductInstruction_tests, 
	stPackCodesDuplicated:= stRejectReasonForOuters_tests.stOuterDuplicatedPackCodesFound, 
	stOuterBarcodeDuplicate:= stRejectReasonForOuters_tests.stOuterBarcodeDuplicate, 
	stOuterDuplicatedPackCodesFound:= stRejectReasonForOuters_tests.stOuterDuplicatedPackCodesFound, 
	stCaseRejectReasons:= stCaseRejectReasons_tests, 
	stCACData:= stCACData_tests, 
	bDone=> bDone_tests, 
	bBusy=> bBusy_tests, 
	bCACValid=> bCACValid_tests, 
	sRejectCode=> sRejectCode_tests, 
	bIsDuplicateOuters=> bIsDuplicateOuter_tests, 
	bIsDuplicatePacks=> bIsDuplicatePacks_tests, 
	bReadyToValidate=> bReadyToValidate_tests, 
	stUpdateCACData=> stUpdateCACData_tests
);

	
AssertEquals_BOOL( Expected	:= FALSE,
			 	   Actual	:= bIsDuplicatePacks_tests, 
			 	   Message	:= 'Duplicated Pack barcode not found');
						

TEST_FINISHED();
END_METHOD

METHOD INTERNAL PackDuplicate01_bIsDuplicatePacksTRUEonPackBarcodeDuplicate
VAR
	fbCase_tests					: FB_CASE_DuplicatCheck;
	
	
	bDone_tests 					: BOOL;
	bBusy_tests						: BOOL;

	bCACValid_tests					: BOOL;
	bIsDuplicateOuter_tests			: BOOL;
	bIsDuplicatePacks_tests			: BOOL;
	
	bReadyToValidate_tests			: BOOL;
	
END_VAR

//Data initialization
TestInit(stCACData:= stCACData_tests, stProductInstruction:= stProductInstruction_tests);

//Change some data for test scenario below
stCACData_tests.Outer[9].PackCode[1] := stCACData_tests.Outer[15].PackCode[5];

	
TcUnit.TEST('PackDuplicate01_bIsDuplicatePacksTRUEonPackBarcodeDuplicate');

fbCase_tests(
	bExecute:= TRUE, 
	stProductInstruction:= stProductInstruction_tests, 
	stPackCodesDuplicated:= stRejectReasonForOuters_tests.stOuterDuplicatedPackCodesFound, 
	stOuterBarcodeDuplicate:= stRejectReasonForOuters_tests.stOuterBarcodeDuplicate, 
	stOuterDuplicatedPackCodesFound:= stRejectReasonForOuters_tests.stOuterDuplicatedPackCodesFound, 
	stCaseRejectReasons:= stCaseRejectReasons_tests, 
	stCACData:= stCACData_tests, 
	bDone=> bDone_tests, 
	bBusy=> bBusy_tests, 
	bCACValid=> bCACValid_tests, 
	sRejectCode=> sRejectCode_tests, 
	bIsDuplicateOuters=> bIsDuplicateOuter_tests, 
	bIsDuplicatePacks=> bIsDuplicatePacks_tests, 
	bReadyToValidate=> bReadyToValidate_tests, 
	stUpdateCACData=> stUpdateCACData_tests
);

	
AssertEquals_BOOL( Expected	:= TRUE,
			 	   Actual	:= bIsDuplicatePacks_tests, 
			 	   Message	:= 'Duplicated Pack barcode not found');
						

TEST_FINISHED();
END_METHOD

METHOD INTERNAL PackDuplicate02_bIsDuplicatePacksTRUEonPackBarcodeDuplicateWithinSameOuter
VAR
	fbCase_tests					: FB_CASE_DuplicatCheck;
	
	
	bDone_tests 					: BOOL;
	bBusy_tests						: BOOL;

	bCACValid_tests					: BOOL;
	bIsDuplicateOuter_tests			: BOOL;
	bIsDuplicatePacks_tests			: BOOL;
	
	bReadyToValidate_tests			: BOOL;
	
END_VAR

//Data initialization
TestInit(stCACData:= stCACData_tests, stProductInstruction:= stProductInstruction_tests);

//Change some data for test scenario below
stCACData_tests.Outer[6].PackCode[1] := stCACData_tests.Outer[6].PackCode[8];

	
TcUnit.TEST('PackDuplicate02_bIsDuplicatePacksTRUEonPackBarcodeDuplicateWithinSameOuter');

fbCase_tests(
	bExecute:= TRUE, 
	stProductInstruction:= stProductInstruction_tests, 
	stPackCodesDuplicated:= stRejectReasonForOuters_tests.stOuterDuplicatedPackCodesFound, 
	stOuterBarcodeDuplicate:= stRejectReasonForOuters_tests.stOuterBarcodeDuplicate, 
	stOuterDuplicatedPackCodesFound:= stRejectReasonForOuters_tests.stOuterDuplicatedPackCodesFound, 
	stCaseRejectReasons:= stCaseRejectReasons_tests, 
	stCACData:= stCACData_tests, 
	bDone=> bDone_tests, 
	bBusy=> bBusy_tests, 
	bCACValid=> bCACValid_tests, 
	sRejectCode=> sRejectCode_tests, 
	bIsDuplicateOuters=> bIsDuplicateOuter_tests, 
	bIsDuplicatePacks=> bIsDuplicatePacks_tests, 
	bReadyToValidate=> bReadyToValidate_tests, 
	stUpdateCACData=> stUpdateCACData_tests
);

	
AssertEquals_BOOL( Expected	:= TRUE,
			 	   Actual	:= bIsDuplicatePacks_tests, 
			 	   Message	:= 'Duplicated Pack barcode not found');
						

TEST_FINISHED();
END_METHOD

METHOD INTERNAL sRejectCodeString01_WrongValueOn1OuterDuplicate
VAR
	fbCase_tests					: FB_CASE_DuplicatCheck;
	
	
	bDone_tests 					: BOOL;
	bBusy_tests						: BOOL;

	bCACValid_tests					: BOOL;
	bIsDuplicateOuter_tests			: BOOL;
	bIsDuplicatePacks_tests			: BOOL;
	
	bReadyToValidate_tests			: BOOL;
	
END_VAR

//Data initialization
TestInit(stCACData:= stCACData_tests, stProductInstruction:= stProductInstruction_tests);

//Change some data for test scenario below
stCACData_tests.Outer[2].Barcode := stCACData_tests.Outer[15].Barcode;

	
TcUnit.TEST('sRejectCodeString01_WrongValueOn1OuterDuplicate');

fbCase_tests(
	bExecute:= TRUE, 
	stProductInstruction:= stProductInstruction_tests, 
	stPackCodesDuplicated:= stRejectReasonForOuters_tests.stOuterDuplicatedPackCodesFound, 
	stOuterBarcodeDuplicate:= stRejectReasonForOuters_tests.stOuterBarcodeDuplicate, 
	stOuterDuplicatedPackCodesFound:= stRejectReasonForOuters_tests.stOuterDuplicatedPackCodesFound, 
	stCaseRejectReasons:= stCaseRejectReasons_tests, 
	stCACData:= stCACData_tests, 
	bDone=> bDone_tests, 
	bBusy=> bBusy_tests, 
	bCACValid=> bCACValid_tests, 
	sRejectCode=> sRejectCode_tests, 
	bIsDuplicateOuters=> bIsDuplicateOuter_tests, 
	bIsDuplicatePacks=> bIsDuplicatePacks_tests, 
	bReadyToValidate=> bReadyToValidate_tests, 
	stUpdateCACData=> stUpdateCACData_tests
);

	
AssertEquals_STRING( Expected	:= 'XXDUP02-15XX',
			 	   		Actual	:= sRejectCode_tests, 
			 	   		Message	:= 'Wrong sRejectCode value on outer duplicate');
						
TEST_FINISHED();
END_METHOD

METHOD INTERNAL sRejectCodeString02_WrongValueOn2PacksDuplicateIn1Outer
VAR
	fbCase_tests					: FB_CASE_DuplicatCheck;
	
	
	bDone_tests 					: BOOL;
	bBusy_tests						: BOOL;

	bCACValid_tests					: BOOL;
	bIsDuplicateOuter_tests			: BOOL;
	bIsDuplicatePacks_tests			: BOOL;
	
	bReadyToValidate_tests			: BOOL;
	
END_VAR

//Data initialization
TestInit(stCACData:= stCACData_tests, stProductInstruction:= stProductInstruction_tests);

//Change some data for test scenario below
stCACData_tests.Outer[12].PackCode[7] := stCACData_tests.Outer[12].PackCode[10];

	
TcUnit.TEST('sRejectCodeString02_WrongValueOn2PacksDuplicateIn1Outer');

fbCase_tests(
	bExecute:= TRUE, 
	stProductInstruction:= stProductInstruction_tests, 
	stPackCodesDuplicated:= stRejectReasonForOuters_tests.stOuterDuplicatedPackCodesFound, 
	stOuterBarcodeDuplicate:= stRejectReasonForOuters_tests.stOuterBarcodeDuplicate, 
	stOuterDuplicatedPackCodesFound:= stRejectReasonForOuters_tests.stOuterDuplicatedPackCodesFound, 
	stCaseRejectReasons:= stCaseRejectReasons_tests, 
	stCACData:= stCACData_tests, 
	bDone=> bDone_tests, 
	bBusy=> bBusy_tests, 
	bCACValid=> bCACValid_tests, 
	sRejectCode=> sRejectCode_tests, 
	bIsDuplicateOuters=> bIsDuplicateOuter_tests, 
	bIsDuplicatePacks=> bIsDuplicatePacks_tests, 
	bReadyToValidate=> bReadyToValidate_tests, 
	stUpdateCACData=> stUpdateCACData_tests
);

	
AssertEquals_STRING( Expected	:= 'XXDUP12(07)-12(10)XX',
			 	   		Actual	:= sRejectCode_tests, 
			 	   		Message	:= 'Wrong sRejectCode value on outer duplicate');
						
TEST_FINISHED();
END_METHOD

METHOD INTERNAL sRejectCodeString03_WrongValueOn2PacksDuplicateIn2Outers
VAR
	fbCase_tests					: FB_CASE_DuplicatCheck;
	
	
	bDone_tests 					: BOOL;
	bBusy_tests						: BOOL;

	bCACValid_tests					: BOOL;
	bIsDuplicateOuter_tests			: BOOL;
	bIsDuplicatePacks_tests			: BOOL;
	
	bReadyToValidate_tests			: BOOL;
	
END_VAR

//Data initialization
TestInit(stCACData:= stCACData_tests, stProductInstruction:= stProductInstruction_tests);

//Change some data for test scenario below
stCACData_tests.Outer[3].PackCode[2] := stCACData_tests.Outer[34].PackCode[6];

	
TcUnit.TEST('sRejectCodeString03_WrongValueOn2PacksDuplicateIn2Outers');

fbCase_tests(
	bExecute:= TRUE, 
	stProductInstruction:= stProductInstruction_tests, 
	stPackCodesDuplicated:= stRejectReasonForOuters_tests.stOuterDuplicatedPackCodesFound, 
	stOuterBarcodeDuplicate:= stRejectReasonForOuters_tests.stOuterBarcodeDuplicate, 
	stOuterDuplicatedPackCodesFound:= stRejectReasonForOuters_tests.stOuterDuplicatedPackCodesFound, 
	stCaseRejectReasons:= stCaseRejectReasons_tests, 
	stCACData:= stCACData_tests, 
	bDone=> bDone_tests, 
	bBusy=> bBusy_tests, 
	bCACValid=> bCACValid_tests, 
	sRejectCode=> sRejectCode_tests, 
	bIsDuplicateOuters=> bIsDuplicateOuter_tests, 
	bIsDuplicatePacks=> bIsDuplicatePacks_tests, 
	bReadyToValidate=> bReadyToValidate_tests, 
	stUpdateCACData=> stUpdateCACData_tests
);

	
AssertEquals_STRING( Expected	:= 'XXDUP03(02)-34(06)XX',
			 	   		Actual	:= sRejectCode_tests, 
			 	   		Message	:= 'Wrong sRejectCode value on outer duplicate');
						
TEST_FINISHED();
END_METHOD

METHOD INTERNAL sRejectCodeString04_WrongValueOnSeveralOutersDuplicate
VAR
	fbCase_tests					: FB_CASE_DuplicatCheck;
	
	
	bDone_tests 					: BOOL;
	bBusy_tests						: BOOL;

	bCACValid_tests					: BOOL;
	bIsDuplicateOuter_tests			: BOOL;
	bIsDuplicatePacks_tests			: BOOL;
	
	bReadyToValidate_tests			: BOOL;
	
END_VAR

//Data initialization
TestInit(stCACData:= stCACData_tests, stProductInstruction:= stProductInstruction_tests);

//Change some data for test scenario below
stCACData_tests.Outer[5].Barcode := stCACData_tests.Outer[39].Barcode;
stCACData_tests.Outer[3].Barcode := stCACData_tests.Outer[25].Barcode;

(************* Now FB returnes last found duplication / is this RIGHT ?***********************)
	
TcUnit.TEST('sRejectCodeString04_WrongValueOnSeveralOutersDuplicate');

fbCase_tests(
	bExecute:= TRUE, 
	stProductInstruction:= stProductInstruction_tests, 
	stPackCodesDuplicated:= stRejectReasonForOuters_tests.stOuterDuplicatedPackCodesFound, 
	stOuterBarcodeDuplicate:= stRejectReasonForOuters_tests.stOuterBarcodeDuplicate, 
	stOuterDuplicatedPackCodesFound:= stRejectReasonForOuters_tests.stOuterDuplicatedPackCodesFound, 
	stCaseRejectReasons:= stCaseRejectReasons_tests, 
	stCACData:= stCACData_tests, 
	bDone=> bDone_tests, 
	bBusy=> bBusy_tests, 
	bCACValid=> bCACValid_tests, 
	sRejectCode=> sRejectCode_tests, 
	bIsDuplicateOuters=> bIsDuplicateOuter_tests, 
	bIsDuplicatePacks=> bIsDuplicatePacks_tests, 
	bReadyToValidate=> bReadyToValidate_tests, 
	stUpdateCACData=> stUpdateCACData_tests
);

	
AssertEquals_STRING( Expected	:= 'XXDUP03-29XX',
			 	   		Actual	:= sRejectCode_tests, 
			 	   		Message	:= 'Wrong sRejectCode value on outer duplicate');
						
TEST_FINISHED();
END_METHOD

METHOD INTERNAL sRejectCodeString05_WrongValueOnSeveralPacksDuplicateInSeveralOuters
VAR
	fbCase_tests					: FB_CASE_DuplicatCheck;
	
	
	bDone_tests 					: BOOL;
	bBusy_tests						: BOOL;

	bCACValid_tests					: BOOL;
	bIsDuplicateOuter_tests			: BOOL;
	bIsDuplicatePacks_tests			: BOOL;
	
	bReadyToValidate_tests			: BOOL;
	
END_VAR

//Data initialization
TestInit(stCACData:= stCACData_tests, stProductInstruction:= stProductInstruction_tests);

//Change some data for test scenario below
stCACData_tests.Outer[3].PackCode[8] 	:= stCACData_tests.Outer[34].PackCode[2];
stCACData_tests.Outer[8].PackCode[7] 	:= stCACData_tests.Outer[15].PackCode[1];
stCACData_tests.Outer[12].PackCode[4] 	:= stCACData_tests.Outer[49].PackCode[10];

	
TcUnit.TEST('sRejectCodeString05_WrongValueOnSeveralPacksDuplicateInSeveralOuters');

fbCase_tests(
	bExecute:= TRUE, 
	stProductInstruction:= stProductInstruction_tests, 
	stPackCodesDuplicated:= stRejectReasonForOuters_tests.stOuterDuplicatedPackCodesFound, 
	stOuterBarcodeDuplicate:= stRejectReasonForOuters_tests.stOuterBarcodeDuplicate, 
	stOuterDuplicatedPackCodesFound:= stRejectReasonForOuters_tests.stOuterDuplicatedPackCodesFound, 
	stCaseRejectReasons:= stCaseRejectReasons_tests, 
	stCACData:= stCACData_tests, 
	bDone=> bDone_tests, 
	bBusy=> bBusy_tests, 
	bCACValid=> bCACValid_tests, 
	sRejectCode=> sRejectCode_tests, 
	bIsDuplicateOuters=> bIsDuplicateOuter_tests, 
	bIsDuplicatePacks=> bIsDuplicatePacks_tests, 
	bReadyToValidate=> bReadyToValidate_tests, 
	stUpdateCACData=> stUpdateCACData_tests
);

	
AssertEquals_STRING( Expected	:= 'XXDUP03(02)-34(06)XX',
			 	   		Actual	:= sRejectCode_tests, 
			 	   		Message	:= 'Wrong sRejectCode value on outer duplicate');
						
TEST_FINISHED();
END_METHOD

METHOD PRIVATE TestInit
VAR_IN_OUT
	stProductInstruction	: ST_PCM_Status;
	stCACData 				: ST_CAC_Data;
END_VAR

VAR	
	rTrigDataInit		: R_TRIG;
	bDataInit			: BOOL;
	iOuter				: INT;
	iPack				: INT;
	sPackNum			: STRING;
	sOuterNum			: STRING;
	sPackCode			: STRING;
END_VAR
MEMSET(ADR(stCACData), 16#00, SIZEOF(stCACData));	

FOR iOuter := 1 TO stProductInstruction.nOutersPerCase DO
		(* Outer number z zerami *)
		sOuterNum := F_StringAddPrefix(INT_TO_STRING(iOuter),2,'0');
		
		(* Write Outers barcodes *)
		stCACData.Outer[iOuter].Barcode    := CONCAT('OUTER', sOuterNum);
		stCACData.Outer[iOuter].OuterCodeStatus := 5;
		
		FOR iPack := 1 TO stProductInstruction.nPacksPerOuter DO
			(* Pack number dwucyfrowy z zerami *)
			sPackNum := F_StringAddPrefix(INT_TO_STRING(iPack),2,'0');			
			(* Sklej pack code *)
			sPackCode := CONCAT(CONCAT('PACK', sPackNum), CONCAT('OUTER', sOuterNum));
			
			(* Write Pack Barcodes *)
			stCACData.Outer[iOuter].PackCode[iPack]			:= sPackCode;
			stCACData.Outer[iOuter].PackCodeStatus[iPack]	:= 5;
			stCACData.Outer[iOuter].PackRejectID[iPack]		:= 0;
			
		END_FOR;
	END_FOR;
END_METHOD

END_FUNCTION_BLOCK

// ---- POUs/TcUnit/FB_CASE_InitialiseData/FB_CASE_InitialiseDataTests.TcPOU
FUNCTION_BLOCK FB_CASE_InitialiseDataTests EXTENDS TcUnit.FB_TestSuite

VAR
	
	(* In/Out test*)		
	stCTDateTime_tests				: ST_SYSTEM_DateTime;	
	stProductInstruction_tests		: ST_PCM_Status;
	stCACData_tests 				: ST_CAC_Data;		
	stRejectReasonsForCase_tets		: ST_RejectReasonsForCase;
		
	sRejectCode_tests				: T_RejectCode;
END_VAR



//==============================================================
//01.Main
//==============================================================
main01_OuterCodeStatus5_NegativeNumberOfOuters();
main02_CaseRejectWrongValuenOpModeBelow6();
main03_DoorRejectIDstatusValueTrue();
main04_CaseRejectWrongValuenOpModeAbove6();
main05_bDoorRejectWrongValueOnDoorReject();

//==============================================================
//02.MasterListCounter
//==============================================================
masterListCounter01_MasterListRestoredCounterWrongNumber01();
masterListCounter02_MasterListRestoredCounterWrongNumber02();
masterListCounter03_MasterListRestoredCounterWrongNumber03();

METHOD INTERNAL main01_OuterCodeStatus5_NegativeNumberOfOuters
VAR
	fbCaseTest				: FB_CASE_InitialiseData;	
	
	bDone_test					: BOOL;
	bBussy_test					: BOOL;
	bDoorReject_test			: BOOL;
	nMasterListCounter_test		: INT;
	bCheckDuplicate_test		: BOOL;

END_VAR

TestInit(stProductInstruction_tests,stCACData_tests);

//Change some data for test scenario below
stCACData_tests.Outer[3].OuterCodeStatus.5 	:= TRUE;
stCACData_tests.Outer[4].OuterCodeStatus.5	:= TRUE;
	
TcUnit.TEST('main01_OuterCodeStatus5_NegativeNumberOfOuters');

fbCaseTest(
	bExecute:= TRUE, 
	stCTDateTime:= stCTDateTime_tests, 
	stDoorGuardReject:= stRejectReasonsForCase_tets.stDoorGuardReject, 
	stProductInstruction:= stProductInstruction_tests, 
	stCACData:= stCACData_tests, 
	bDone=> bDone_test, 
	bBusy=> bBussy_test, 
	bDoorReject=> bDoorReject_test, 
	sRejectCode=> sRejectCode_tests, 
	nMasterListCounter=> nMasterListCounter_test, 
	bCheckDuplicates=> bCheckDuplicate_test
	
	);

	AssertEquals_INT(	Expected:= -3, 
						Actual:= stCACData_tests.NumberOfOuters, 
						Message:= 'Wrong NumberOfOuters parameter (Val Index)');
						
						


TEST_FINISHED();
END_METHOD

METHOD INTERNAL main02_CaseRejectWrongValuenOpModeBelow6
VAR
	fbCaseTest				: FB_CASE_InitialiseData;	
	
	bDone_test					: BOOL;
	bBussy_test					: BOOL;
	bDoorReject_test			: BOOL;
	nMasterListCounter_test		: INT;
	bCheckDuplicate_test		: BOOL;
	
	sRejectCodeTemp				: T_RejectCode;
	
END_VAR

TestInit(stProductInstruction_tests,stCACData_tests);

//Change some data for test scenario below
sRejectCodeTemp := '';
stProductInstruction_tests.nOpMode	:= 5;


fbCaseTest(
	bExecute:= TRUE, 
	stCTDateTime:= stCTDateTime_tests, 
	stDoorGuardReject:= stRejectReasonsForCase_tets.stDoorGuardReject, 
	stProductInstruction:= stProductInstruction_tests, 
	stCACData:= stCACData_tests, 
	bDone=> bDone_test, 
	bBusy=> bBussy_test, 
	bDoorReject=> bDoorReject_test, 
	sRejectCode=> sRejectCode_tests, 
	nMasterListCounter=> nMasterListCounter_test, 
	bCheckDuplicates=> bCheckDuplicate_test
	
	);

TcUnit.TEST('main02_CaseRejectWrongValue');


						
	AssertEquals_STRING(Expected := TO_STRING(sRejectCodeTemp),
                    Actual := TO_STRING(sRejectCode_tests),
                    Message := 'Values of CaseRejectCode differ');

TEST_FINISHED();
END_METHOD

METHOD INTERNAL main03_DoorRejectIDstatusValueTrue
VAR
	fbCaseTest				: FB_CASE_InitialiseData;	
	
	bDone_test					: BOOL;
	bBussy_test					: BOOL;
	bDoorReject_test			: BOOL;
	nMasterListCounter_test		: INT;
	bCheckDuplicate_test		: BOOL;
	
END_VAR

TestInit(stProductInstruction_tests,stCACData_tests);

//Change some data for test scenario below
stRejectReasonsForCase_tets.stDoorGuardReject.nRejectID := 311;
stCACData_tests.CaseRejectID := 311;
(* PassThrough, PrePrintedLabel or PrintApply mode active *)
stProductInstruction_tests.nOpMode := 6;


fbCaseTest(
	bExecute:= TRUE, 
	stCTDateTime:= stCTDateTime_tests, 
	stDoorGuardReject:= stRejectReasonsForCase_tets.stDoorGuardReject, 
	stProductInstruction:= stProductInstruction_tests, 
	stCACData:= stCACData_tests, 
	bDone=> bDone_test, 
	bBusy=> bBussy_test, 
	bDoorReject=> bDoorReject_test, 
	sRejectCode=> sRejectCode_tests, 
	nMasterListCounter=> nMasterListCounter_test, 
	bCheckDuplicates=> bCheckDuplicate_test
	
	);

TcUnit.TEST('main03_DoorRejectIDstatusValueTrue');


						
	AssertEquals_BOOL(	Expected := TRUE, 
						Actual:= bDoorReject_test, 
						Message:= 'bDoorReject wrong value');

TEST_FINISHED();
END_METHOD

METHOD INTERNAL main04_CaseRejectWrongValuenOpModeAbove6
VAR
	fbCaseTest				: FB_CASE_InitialiseData;	
	
	bDone_test					: BOOL;
	bBussy_test					: BOOL;
	bDoorReject_test			: BOOL;
	nMasterListCounter_test		: INT;
	bCheckDuplicate_test		: BOOL;
	
	sRejectCodeTemp				: T_RejectCode;
	
END_VAR

TestInit(stProductInstruction_tests,stCACData_tests);

//Change some data for test scenario below
sRejectCodeTemp := 'OK';
stProductInstruction_tests.nOpMode	:= 9;


fbCaseTest(
	bExecute:= TRUE, 
	stCTDateTime:= stCTDateTime_tests, 
	stDoorGuardReject:= stRejectReasonsForCase_tets.stDoorGuardReject, 
	stProductInstruction:= stProductInstruction_tests, 
	stCACData:= stCACData_tests, 
	bDone=> bDone_test, 
	bBusy=> bBussy_test, 
	bDoorReject=> bDoorReject_test, 
	sRejectCode=> sRejectCode_tests, 
	nMasterListCounter=> nMasterListCounter_test, 
	bCheckDuplicates=> bCheckDuplicate_test
	
	);

TcUnit.TEST('main04_CaseRejectWrongValuenOpModeAbove6');


						
	AssertEquals_STRING(Expected := TO_STRING(sRejectCodeTemp),
                    Actual := TO_STRING(sRejectCode_tests),
                    Message := 'Values of CaseRejectCode differ');

TEST_FINISHED();
END_METHOD

METHOD INTERNAL main05_bDoorRejectWrongValueOnDoorReject
VAR
	fbCaseTest				: FB_CASE_InitialiseData;	
	
	bDone_test					: BOOL;
	bBussy_test					: BOOL;
	bDoorReject_test			: BOOL;
	nMasterListCounter_test		: INT;
	bCheckDuplicate_test		: BOOL;
	
	
END_VAR

TestInit(stProductInstruction_tests,stCACData_tests);

//Change some data for test scenario below
stCACData_tests.CaseRejectID := stRejectReasonsForCase_tets.stDoorGuardReject.nRejectID;
stProductInstruction_tests.nOpMode := 5;


fbCaseTest(
	bExecute:= TRUE, 
	stCTDateTime:= stCTDateTime_tests, 
	stDoorGuardReject:= stRejectReasonsForCase_tets.stDoorGuardReject, 
	stProductInstruction:= stProductInstruction_tests, 
	stCACData:= stCACData_tests, 
	bDone=> bDone_test, 
	bBusy=> bBussy_test, 
	bDoorReject=> bDoorReject_test, 
	sRejectCode=> sRejectCode_tests, 
	nMasterListCounter=> nMasterListCounter_test, 
	bCheckDuplicates=> bCheckDuplicate_test
	
	);

TcUnit.TEST('main05_bDoorRejectWrongValueOnDoorReject');

	AssertEquals_BOOL(Expected  := TRUE,
                  	  Actual 	:= bDoorReject_test,
                   	  Message 	:= 'bDoorReject wrong value');

TEST_FINISHED();
END_METHOD

METHOD INTERNAL masterListCounter01_MasterListRestoredCounterWrongNumber01
VAR
	fbCaseTest					: FB_CASE_InitialiseData;	
	
	bDone_test					: BOOL;
	bBussy_test					: BOOL;
	bDoorReject_test			: BOOL;
	nMasterListCounter_test		: INT;
	bCheckDuplicate_test		: BOOL;

	
END_VAR

TestInit(stProductInstruction_tests,stCACData_tests);

//Change some data for test scenario below	
stCACData_tests.Outer[1].OuterMasterListRestored	:= TRUE;
stCACData_tests.Outer[25].OuterMasterListRestored	:= TRUE;
stCACData_tests.Outer[49].OuterMasterListRestored	:= TRUE;
//outers in case 50, table size 70
stCACData_tests.Outer[67].OuterMasterListRestored	:= TRUE;

fbCaseTest(
	bExecute:= TRUE, 
	stCTDateTime:= stCTDateTime_tests, 
	stDoorGuardReject:= stRejectReasonsForCase_tets.stDoorGuardReject, 
	stProductInstruction:= stProductInstruction_tests, 
	stCACData:= stCACData_tests, 
	bDone=> bDone_test, 
	bBusy=> bBussy_test, 
	bDoorReject=> bDoorReject_test, 
	sRejectCode=> sRejectCode_tests, 
	nMasterListCounter=> nMasterListCounter_test, 
	bCheckDuplicates=> bCheckDuplicate_test
	
	);

TcUnit.TEST('masterListCounter01_MasterListRestoredCounterWrongNumber01');



	AssertEquals_INT(	Expected:= 3, 
						Actual:= nMasterListCounter_test, 
						Message:= 'Wrong count of restored outer');
						
	AssertEquals_BOOL(	Expected := TRUE, 
						Actual:= stCACData_tests.Outer[49].OuterMasterListRestored, 
						Message:= 'Outer master list restored status wrong value');

TEST_FINISHED();
END_METHOD

METHOD INTERNAL masterListCounter02_MasterListRestoredCounterWrongNumber02
VAR
	fbCaseTest					: FB_CASE_InitialiseData;	
	
	bDone_test					: BOOL;
	bBussy_test					: BOOL;
	bDoorReject_test			: BOOL;
	nMasterListCounter_test		: INT;
	bCheckDuplicate_test		: BOOL;

	
END_VAR

TestInit(stProductInstruction_tests,stCACData_tests);

//Change some data for test scenario below	
stCACData_tests.Outer[9].OuterMasterListRestored	:= TRUE;
stCACData_tests.Outer[15].OuterMasterListRestored	:= TRUE;
stCACData_tests.Outer[18].OuterMasterListRestored	:= TRUE;
stCACData_tests.Outer[21].OuterMasterListRestored	:= TRUE;
stCACData_tests.Outer[27].OuterMasterListRestored	:= TRUE;
stCACData_tests.Outer[30].OuterMasterListRestored	:= TRUE;
stCACData_tests.Outer[32].OuterMasterListRestored	:= TRUE;
stCACData_tests.Outer[38].OuterMasterListRestored	:= TRUE;
stCACData_tests.Outer[45].OuterMasterListRestored	:= TRUE;
stCACData_tests.Outer[46].OuterMasterListRestored	:= TRUE;
stCACData_tests.Outer[50].OuterMasterListRestored	:= TRUE;

//outers in case 50, table size 70
stCACData_tests.Outer[67].OuterMasterListRestored	:= TRUE;

fbCaseTest(
	bExecute:= TRUE, 
	stCTDateTime:= stCTDateTime_tests, 
	stDoorGuardReject:= stRejectReasonsForCase_tets.stDoorGuardReject, 
	stProductInstruction:= stProductInstruction_tests, 
	stCACData:= stCACData_tests, 
	bDone=> bDone_test, 
	bBusy=> bBussy_test, 
	bDoorReject=> bDoorReject_test, 
	sRejectCode=> sRejectCode_tests, 
	nMasterListCounter=> nMasterListCounter_test, 
	bCheckDuplicates=> bCheckDuplicate_test
	
	);

TcUnit.TEST('masterListCounter02_MasterListRestoredCounterWrongNumber02');



	AssertEquals_INT(	Expected:= 11, 
						Actual:= nMasterListCounter_test, 
						Message:= 'Wrong count of restored outer');

TEST_FINISHED();
END_METHOD

METHOD INTERNAL masterListCounter03_MasterListRestoredCounterWrongNumber03
VAR
	fbCaseTest					: FB_CASE_InitialiseData;	
	
	bDone_test					: BOOL;
	bBussy_test					: BOOL;
	bDoorReject_test			: BOOL;
	nMasterListCounter_test		: INT;
	bCheckDuplicate_test		: BOOL;

	
END_VAR

TestInit(stProductInstruction_tests,stCACData_tests);

//Change some data for test scenario below	
stCACData_tests.Outer[4].OuterMasterListRestored	:= FALSE;
stCACData_tests.Outer[23].OuterMasterListRestored	:= TRUE;
stCACData_tests.Outer[69].OuterMasterListRestored	:= TRUE;

//outers in case 50, table size 70
stCACData_tests.Outer[67].OuterMasterListRestored	:= TRUE;

fbCaseTest(
	bExecute:= TRUE, 
	stCTDateTime:= stCTDateTime_tests, 
	stDoorGuardReject:= stRejectReasonsForCase_tets.stDoorGuardReject, 
	stProductInstruction:= stProductInstruction_tests, 
	stCACData:= stCACData_tests, 
	bDone=> bDone_test, 
	bBusy=> bBussy_test, 
	bDoorReject=> bDoorReject_test, 
	sRejectCode=> sRejectCode_tests, 
	nMasterListCounter=> nMasterListCounter_test, 
	bCheckDuplicates=> bCheckDuplicate_test
	
	);

TcUnit.TEST('masterListCounter03_MasterListRestoredCounterWrongNumber03');



	AssertEquals_INT(	Expected:= 1, 
						Actual:= nMasterListCounter_test, 
						Message:= 'Wrong count of restored outer');

TEST_FINISHED();
END_METHOD

METHOD PRIVATE TestInit
VAR_IN_OUT
	stProductInstruction	: ST_PCM_Status;
	stCACData 				: ST_CAC_Data;	(* Case Queue *)
END_VAR

VAR	
	(* Init function/method declarations*)
	rTrigDataInit		: R_TRIG;
	bDataInit			: BOOL;
	iOuter				: INT;
	iPack				: INT;
	sPackNum			: STRING;
	sOuterNum			: STRING;
	sPackCode			: STRING;
END_VAR
MEMSET(ADR(stCACData), 16#00, SIZEOF(stCACData));	
	
stProductInstruction.nOutersPerCase 	:= 50;
stProductInstruction.nPacksPerOuter		:= 10;
stProductInstruction.nOpMode			:= 11;
stProductInstruction.sRetailSKU			:= '1234567';
stProductInstruction.nAcceptanceLevel 	:= 10;


stCACData.NumberOfOuters			:= stProductInstruction.nOutersPerCase;
stCACData.CodingAndTrackingMode		:= stProductInstruction.nOpMode;
stCACData.RetailSKU					:= stProductInstruction.sRetailSKU;

FOR iOuter := 1 TO stProductInstruction.nOutersPerCase DO
	(* Outer number with prefix '0' *)
	sOuterNum := F_StringAddPrefix(INT_TO_STRING(iOuter),2,'0');

	stCACData.Outer[iOuter].Barcode    				:= CONCAT('OUTER', sOuterNum);
	stCACData.Outer[iOuter].NumberOfPacks 			:= stProductInstruction.nPacksPerOuter;
	stCACData.Outer[iOuter].NumberOfLinkedPacks 	:= stProductInstruction.nPacksPerOuter;
	stCACData.Outer[iOuter].AcceptanceLevel 		:= stProductInstruction.nAcceptanceLevel;
	stCACData.Outer[iOuter].CodingAndTrackingMode	:= stProductInstruction.nOpMode;
	stCACData.Outer[iOuter].OuterRejectCode			:= 'OK';

	FOR iPack := 1 TO stProductInstruction.nPacksPerOuter DO
		(* Pack number dwucyfrowy z zerami *)
		sPackNum := F_StringAddPrefix(INT_TO_STRING(iPack),2,'0');			
		(* Sklej pack code *)
		sPackCode := CONCAT(CONCAT('PACK', sPackNum), CONCAT('OUTER', sOuterNum));
		
		(* Write Pack Barcodes / Data*)
		stCACData.Outer[iOuter].PackCode[iPack]				:= sPackCode;
		stCACData.Outer[iOuter].PackCodeStatus[iPack]		:= 5;
		stCACData.Outer[iOuter].PackRejectID[iPack]			:= 0;			
		stCACData.Outer[iOuter].PackRejectCode[iPack]		:= 'OK';			
		stCACData.Outer[iOuter].PackCodeStatus[iPack].5 	:= TRUE;
		
		
		IF iPack = 1 THEN
			stCACData.Outer[iOuter].AggregationCodes[1]	:= stCACData.Outer[iOuter].PackCode[iPack];
		END_IF
		IF iPack = 2 THEN
			stCACData.Outer[iOuter].AggregationCodes[2]	:= stCACData.Outer[iOuter].PackCode[iPack];
		END_IF
	END_FOR
END_FOR
END_METHOD

END_FUNCTION_BLOCK

// ---- POUs/TcUnit/FB_CASE_FinaliseDataTests/FB_CASE_FinaliseDataTests.TcPOU
FUNCTION_BLOCK FB_CASE_FinaliseDataTests EXTENDS TcUnit.FB_TestSuite

VAR
	
	(* In/Out test*)
	stProductInstruction_tests					: ST_PCM_Status;
	stOuterBarcodeDuplicate_tests				: ST_RejectItems;
	stOuterDuplicatedPackCodesFound_tests		: ST_RejectItems;
	stCaseRejectReasons_tests					: ST_RejectReasonsForCase;		
	stRejectReasonForOuters_tests				: ST_RejectReasonsForOuter;	
	stRejectReasonForPacks_tests				: ST_RejectReasonsForPack;		
	stCodeInfo_Outer_tests						: ST_CodeInfo;
	
	stCACData_tests 							: ST_CAC_Data;	
	stUpdateCACData_tests						: ST_CAC_Data;	
	sRejectCode_tests							: T_MaxString;
	stCACDataHMI_tests							: ST_HMI_CAC_Data;
	sCaseContent_tests							: T_LongSTRING;
	
	
END_VAR


stProductInstruction_tests.nOutersPerCase			:= 50;
stProductInstruction_tests.nPacksPerOuter 			:= 10;


stCACData_tests.NumberOfOuters							:= stProductInstruction_tests.nOutersPerCase;
stCACData_tests.CaseRejectCode							:= 'OK';
stCodeInfo_Outer_tests.nEntireLength					:= 7;
stCodeInfo_Outer_tests.stSerialCode.nCodeStartPos 		:= 1;
stCodeInfo_Outer_tests.stSerialCode.nCodeLength 		:= 7;

//==============================================================
//01.Main
//==============================================================
main01_FBExecuted_bDoneTRUE();
main02_bCACValidTrueOnValidData();
main03_bCACInvalidFalseOnValidData();
main04_bCACInvalidTrueOnInvalidData();
main05_bCACValidFalseOnInvalidData();
main06_FBnotExecuted_bDoneFALSE();
main07_FBExecuted_bReadyToValidateFALSE();
main08_FBExecuted_bCheckDuplicatesFALSEonOuterDuplicates();


//==============================================================
//02.CaseContenr	
//==============================================================
caseContent01_sCaseContentValueValid();
caseContent02_sCaseContentValueToShort();
caseContent03_sCaseContentValueToLong();


//==============================================================
//03. DataHMI
//==============================================================
dataHMI01_CaseBarcodeNotOkOnValidData();
dataHMI02_CaseBarcodeOkOnInalidData();
dataHMI03_OuterBarcodeOkOnInalidData();
dataHMI04_OuterBarcodeNotOkOnValidData();
dataHMI05_PackBarcodeOkOnInvalidData();
dataHMI06_PackBarcodeNotOkOnValidData();

METHOD INTERNAL caseContent01_sCaseContentValueValid
VAR
	fbCase_tests		: FB_CASE_FinaliseData;
	
	bDoorReject			: BOOL;	
	bDone 				: BOOL;
	bBusy				: BOOL;

	bCACValid			: BOOL;
	bCACInvalid			: BOOL;

	bCheckDuplicates	: BOOL;
	bReadyToValidate	: BOOL;
	
	minLength			: UDINT;
	nCompare			: DINT;
	sCaseContentTEMP	: T_LongSTRING; 
		
END_VAR

//Data initialization
TestInit(stCACData:= stCACData_tests, stProductInstruction:= stProductInstruction_tests);

//Change some data for test scenario below
sCaseContentTEMP := ' [50]:   OUTER01   OUTER02   OUTER03   OUTER04   OUTER05   OUTER06   OUTER07   OUTER08   OUTER09   OUTER10   OUTER11   OUTER12   OUTER13   OUTER14   OUTER15   OUTER16   OUTER17   OUTER18   OUTER19   OUTER20   OUTER21   OUTER22   OUTER23   OUTER24   OUTER25   OUTER26   OUTER27   OUTER28   OUTER29   OUTER30   OUTER31   OUTER32   OUTER33   OUTER34   OUTER35   OUTER36   OUTER37   OUTER38   OUTER39   OUTER40   OUTER41   OUTER42   OUTER43   OUTER44   OUTER45   OUTER46   OUTER47   OUTER48   OUTER49   OUTER50';

	
TcUnit.TEST('caseContent01_sCaseContentValueValid');

fbCase_tests(
	bExecute:= TRUE, 
	bDoorReject:= bDoorReject, 
	stDoorGuardReject:= stCaseRejectReasons_tests.stDoorGuardReject, 
	stProductInstruction:= stProductInstruction_tests, 
	stCodeInfo_Outer:= stCodeInfo_Outer_tests, 
	stCACData:= stCACData_tests, 
	stCACDataHMI:= stCACDataHMI_tests, 
	bDone=> bDone, 
	bBusy=> bBusy, 
	bCACValid=> bCACValid, 
	bCACInvalid=> bCACInvalid, 
	bCheckDuplicates=> bCheckDuplicates, 
	bReadyToValidate=> bReadyToValidate, 
	sRejectCode=> sRejectCode_tests, 
	sCaseContent=> sCaseContent_tests);


minLength 	:= MIN(TO_UDINT(LEN(sCaseContentTEMP)), TO_UDINT(LEN(sCaseContent_tests)));
nCompare	:= MEMCMP(pBuf1:= ADR(sCaseContentTEMP), pBuf2:= ADR(sCaseContent_tests), n:= minLength);
	
AssertEquals_DINT(Expected := 0,
                  Actual := nCompare,
                  Message := 'Value of sCaseContent wrong');
						

TEST_FINISHED();
END_METHOD

METHOD INTERNAL caseContent02_sCaseContentValueToShort
VAR
	fbCase_tests		: FB_CASE_FinaliseData;
	
	bDoorReject			: BOOL;	
	bDone 				: BOOL;
	bBusy				: BOOL;

	bCACValid			: BOOL;
	bCACInvalid			: BOOL;

	bCheckDuplicates	: BOOL;
	bReadyToValidate	: BOOL;
	
	minLength			: UDINT;
	nCompare			: DINT;
	sCaseContentTEMP	: T_LongSTRING; 
		
END_VAR

//Data initialization
TestInit(stCACData:= stCACData_tests, stProductInstruction:= stProductInstruction_tests);

//Change some data for test scenario below
sCaseContentTEMP := ' [50]:   OUTER02   OUTER03   OUTER04   OUTER05   OUTER06   OUTER07   OUTER08   OUTER09   OUTER10   OUTER11   OUTER12   OUTER13   OUTER14   OUTER15   OUTER16   OUTER17   OUTER18   OUTER19   OUTER20   OUTER21   OUTER22   OUTER23   OUTER24   OUTER25   OUTER26   OUTER27   OUTER28   OUTER29   OUTER30   OUTER31   OUTER32   OUTER33   OUTER34   OUTER35   OUTER36   OUTER37   OUTER38   OUTER39   OUTER40   OUTER41   OUTER42   OUTER43   OUTER44   OUTER45   OUTER46   OUTER47   OUTER48   OUTER49   OUTER50';

	
TcUnit.TEST('caseContent02_sCaseContentValueToShort');

fbCase_tests(
	bExecute:= TRUE, 
	bDoorReject:= bDoorReject, 
	stDoorGuardReject:= stCaseRejectReasons_tests.stDoorGuardReject, 
	stProductInstruction:= stProductInstruction_tests, 
	stCodeInfo_Outer:= stCodeInfo_Outer_tests, 
	stCACData:= stCACData_tests, 
	stCACDataHMI:= stCACDataHMI_tests, 
	bDone=> bDone, 
	bBusy=> bBusy, 
	bCACValid=> bCACValid, 
	bCACInvalid=> bCACInvalid, 
	bCheckDuplicates=> bCheckDuplicates, 
	bReadyToValidate=> bReadyToValidate, 
	sRejectCode=> sRejectCode_tests, 
	sCaseContent=> sCaseContent_tests);


minLength 	:= MAX(TO_UDINT(LEN(sCaseContentTEMP)), TO_UDINT(LEN(sCaseContent_tests)));
nCompare	:= MEMCMP(pBuf1:= ADR(sCaseContentTEMP), pBuf2:= ADR(sCaseContent_tests), n:= minLength);
	
AssertEquals_DINT(Expected := 1,
                  Actual := nCompare,
                  Message := 'Value of sCaseContent wrong');
						

TEST_FINISHED();
END_METHOD

METHOD INTERNAL caseContent03_sCaseContentValueToLong
VAR
	fbCase_tests		: FB_CASE_FinaliseData;
	
	bDoorReject			: BOOL;	
	bDone 				: BOOL;
	bBusy				: BOOL;

	bCACValid			: BOOL;
	bCACInvalid			: BOOL;

	bCheckDuplicates	: BOOL;
	bReadyToValidate	: BOOL;
	
	minLength			: UDINT;
	nCompare			: DINT;
	sCaseContentTEMP	: T_LongSTRING; 
		
END_VAR

//Data initialization
TestInit(stCACData:= stCACData_tests, stProductInstruction:= stProductInstruction_tests);

//Change some data for test scenario below
sCaseContentTEMP := ' [50]:   OUTER51   OUTER01   OUTER02   OUTER03   OUTER04   OUTER05   OUTER06   OUTER07   OUTER08   OUTER09   OUTER10   OUTER11   OUTER12   OUTER13   OUTER14   OUTER15   OUTER16   OUTER17   OUTER18   OUTER19   OUTER20   OUTER21   OUTER22   OUTER23   OUTER24   OUTER25   OUTER26   OUTER27   OUTER28   OUTER29   OUTER30   OUTER31   OUTER32   OUTER33   OUTER34   OUTER35   OUTER36   OUTER37   OUTER38   OUTER39   OUTER40   OUTER41   OUTER42   OUTER43   OUTER44   OUTER45   OUTER46   OUTER47   OUTER48   OUTER49   OUTER50';

	
TcUnit.TEST('caseContent03_sCaseContentValueToLong');

fbCase_tests(
	bExecute:= TRUE, 
	bDoorReject:= bDoorReject, 
	stDoorGuardReject:= stCaseRejectReasons_tests.stDoorGuardReject, 
	stProductInstruction:= stProductInstruction_tests, 
	stCodeInfo_Outer:= stCodeInfo_Outer_tests, 
	stCACData:= stCACData_tests, 
	stCACDataHMI:= stCACDataHMI_tests, 
	bDone=> bDone, 
	bBusy=> bBusy, 
	bCACValid=> bCACValid, 
	bCACInvalid=> bCACInvalid, 
	bCheckDuplicates=> bCheckDuplicates, 
	bReadyToValidate=> bReadyToValidate, 
	sRejectCode=> sRejectCode_tests, 
	sCaseContent=> sCaseContent_tests);


minLength 	:= MIN(TO_UDINT(LEN(sCaseContentTEMP)), TO_UDINT(LEN(sCaseContent_tests)));
nCompare	:= MEMCMP(pBuf1:= ADR(sCaseContentTEMP), pBuf2:= ADR(sCaseContent_tests), n:= minLength);
	
AssertEquals_DINT(Expected := -1,
                  Actual := nCompare,
                  Message := 'Value of sCaseContent wrong');
						

TEST_FINISHED();
END_METHOD

METHOD INTERNAL dataHMI01_CaseBarcodeNotOkOnValidData
VAR
	fbCase_tests		: FB_CASE_FinaliseData;
	
	bDoorReject			: BOOL;	
	bDone 				: BOOL;
	bBusy				: BOOL;

	bCACValid			: BOOL;
	bCACInvalid			: BOOL;

	bCheckDuplicates	: BOOL;
	bReadyToValidate	: BOOL;
	
	sTempCaseBarcode		: T_CASE_Barcode;
	bEqualCaseBarcodeCheck	: BOOL;			
		
END_VAR

//Data initialization
TestInit(stCACData:= stCACData_tests, stProductInstruction:= stProductInstruction_tests);

//Change some data for test scenario below
stCACData_tests.CaseRejectCode := 'OK'; // data OK
stCACData_tests.Barcode := 'CaseBarcode'; // dummyValue
sTempCaseBarcode := F_CONCAT3(stCACData_tests.Barcode,'(999)','1');
	
TcUnit.TEST('dataHMI01_CaseBarcodeNotOkOnValidData');

